// Mitsubishi GX Works2 project: A02_20251220_0   PLC: Q03UDV

TYPE Auto_Data : STRUCT
  Auto_Step : INT;  (* 自动流程字 *)
  Error_Code : INT;  (* 错误码 *)
  Task_Type : WORD;  (* 任务类型 *)
  Start_Row : INT;  (* 起点排 *)
  Start_Column : INT;  (* 起点列 *)
  Start_Layer : INT;  (* 起点层 *)
  End_Row : INT;  (* 终点排 *)
  End_Column : INT;  (* 终点列 *)
  End_Layer : INT;  (* 终点层 *)
  Picking_Station_No : INT;  (* 入库台编号 *)
  Placing_Station_No : INT;  (* 出库台编号 *)
  Task_Status : WORD;  (* 任务状态 *)
  Current_Task_ID : DWORD;  (* 当前任务ID *)
  Total_Number_Tasks : DINT;  (* 任务执行总次数 *)
  Stacker_Status : WORD;  (* 堆垛机状态 *)
  X_Current_Actual_Position : REAL;  (* X轴行走当前实际位置 *)
  Y_Current_Actual_Position : REAL;  (* Y轴升降当前实际位置 *)
  Z_Current_Actual_Position : REAL;  (* Z轴货叉当前实际位置 *)
  X_Current_Actual_Speed : REAL;  (* X轴行走当前实际速度 *)
  Y_Current_Actual_Speed : REAL;  (* Y轴升降当前实际速度 *)
  Z_Current_Actual_Speed : REAL;  (* Z轴货叉当前实际速度 *)
END_STRUCT END_TYPE

TYPE Axle_Data : STRUCT
  Auto_Target_Position : REAL;  (* Auto_目标位置 *)
  Auto_Positioning_Speed : REAL;  (* Auto_定位速度 *)
  Auto_Enable_Location : ARRAY [0..15] OF BOOL;  (* Auto_开启定位 *)
  Auto_Position_Reached : BOOL;  (* Auto_位置到达 *)
  Jog_Forward : BOOL;  (* 点动正转 *)
  Jog_Reverse : BOOL;  (* 点动反转 *)
  Forward_Enable : BOOL;  (* 正转允许 *)
  Reverse_Enable : BOOL;  (* 反转允许 *)
  o_wdCurrentPosition_F : REAL;  (* 当前位置 *)
  o_wdCurrentSpeed_F : REAL;  (* 当前速度 *)
  i_wdTargetPosition_F : REAL;  (* 目标位置 *)
  i_wdTargetVelocity_F : REAL;  (* 定位速度 *)
END_STRUCT END_TYPE

TYPE Pos : STRUCT
  X_Position : REAL;
  Y_Position : REAL;
  Z_Position : REAL;
END_STRUCT END_TYPE

TYPE Axle_attribute : STRUCT
  Motor_Actual_Position : REAL;  (* 电机实际位置 *)
  Position_Difference : REAL;  (* 位置差 *)
  Position_Reached : BOOL;  (* 位置到达 *)
END_STRUCT END_TYPE

TYPE Fork_Alarm : STRUCT
  Fork_Left_collapse_Alarm1 : BOOL;  (* 货叉左侧坍塌报警1 *)
  Fork_Left_collapse_Alarm2 : BOOL;  (* 货叉左侧坍塌报警2 *)
  Fork_Left_Width_Alarm1 : BOOL;  (* 货叉左超宽报警1 *)
  Fork_Left_Width_Alarm2 : BOOL;  (* 货叉左超宽报警2 *)
  Fork_Left_Height_Alarm : BOOL;  (* 货叉左侧超高报警 *)
  Fork_Right_collapse_Alarm1 : BOOL;  (* 货叉右侧坍塌报警1 *)
  Fork_Right_collapse_Alarm2 : BOOL;  (* 货叉右侧坍塌报警2 *)
  Fork_Right_Width_Alarm1 : BOOL;  (* 货叉右超宽报警1 *)
  Fork_Right_Width_Alarm2 : BOOL;  (* 货叉右超宽报警2 *)
  Fork_Right_Height_Alarm : BOOL;  (* 货叉右侧超高报警 *)
END_STRUCT END_TYPE

TYPE Sew_Write : STRUCT
  Control_Character : INT;  (* 控制字 *)
  Rated_Speed : INT;  (* 额定速度 *)
  Acceleration : INT;  (* 加速度 *)
  Deceleration : INT;  (* 减速度 *)
  Virtual_Input_Port : INT;  (* 虚拟输入端 *)
  Set_Mode : INT;  (* 设定应用模式 *)
  Target_Position : DINT;  (* 目标位置 *)
END_STRUCT END_TYPE

TYPE Sew_Read : STRUCT
  Status_Character : INT;  (* 状态字 *)
  Actual_Speed : INT;  (* 实际速度 *)
  Main_Status_Fault : WORD;  (* 状态主故障 *)
  Actual_Torque : INT;  (* 实际扭矩 *)
  Digital_Input_Port : INT;  (* 数字输入端 *)
  Actual_Mode : INT;  (* 实际应用模式 *)
  Actual_Position : DINT;  (* 实际位置 *)
END_STRUCT END_TYPE

TYPE Wcs_Data : STRUCT
  Task_Type : WORD;  (* 任务类型 *)
  Task_ID : DWORD;  (* 任务ID *)
  Start_Row : INT;  (* 起点排 *)
  Start_Column : INT;  (* 起点列 *)
  Start_Layer : INT;  (* 起点层 *)
  End_Row : INT;  (* 终点排 *)
  End_Column : INT;  (* 终点列 *)
  End_Layer : INT;  (* 终点层 *)
  Picking_Station_No : INT;  (* 入库台编号 *)
  Placing_Station_No : INT;  (* 出库台编号 *)
END_STRUCT END_TYPE

TYPE station_Status : STRUCT
  LoadGoods_Enable : BOOL;  (* 允许入库 *)
  UnLoadGoods_Enable : BOOL;  (* 允许出库 *)
END_STRUCT END_TYPE

TYPE manual_data : STRUCT
  X_ManualStart_Position : BOOL;  (* X轴单独定位 *)
  Y_ManualStart_Position : BOOL;  (* Y轴单独定位 *)
  Z_ManualStart_Position : BOOL;  (* Z轴单独定位 *)
  Position_Coords_Switch : BOOL;  (* 位置库位坐标切换 *)
  X_ManualPosition : REAL;  (* X轴定位位置 *)
  Y_ManualPosition : REAL;  (* Y轴定位位置 *)
  Z_ManualPosition : REAL;  (* Z轴定位位置 *)
  X_Manual_Column : INT;  (* X库位列 *)
  Y_Manual_Layer : INT;  (* Y库位层 *)
  X_ManualPosition_Assist : REAL;  (* X轴定位位置辅助 *)
  Y_ManualPosition_Assist : REAL;  (* Y轴定位位置辅助 *)
  Z_ManualPosition_Assist : REAL;  (* Z轴定位位置辅助 *)
  X_Manual_Column_Assist : INT;  (* X库位列辅助 *)
  Y_Manual_Layer_Assist : INT;  (* Y库位层辅助 *)
END_STRUCT END_TYPE

TYPE DInput : STRUCT
  AO2Safety_Circuit1 : BOOL;  (* AO2安全回路1 *)
  AO2Safety_Circuit2 : BOOL;  (* AO2安全回路2 *)
  Maintain_Run : BOOL;  (* 检修运行 *)
  Alarm_Reset : BOOL;  (* 故障复位 *)
  Admin : BOOL;  (* 管理者 *)
  Spare : BOOL;  (* 备用 *)
  Forward_Laser_Stop : BOOL;  (* 行走前方避障信号 *)
  Forward_Laser_Alarm : BOOL;  (* 行走前方避障故障 *)
  Reverse_Laser_Stop : BOOL;  (* 行走后方避障信号 *)
  Reverse_Laser_Alarm : BOOL;  (* 行走后方避障故障 *)
  Spare1 : BOOL;  (* 备用1 *)
  Spare2 : BOOL;  (* 备用2 *)
  Walk_Forward_TO_Pos : BOOL;  (* 行走前方限位 *)
  Walk_Reverse_TO_Pos : BOOL;  (* 行走后方限位 *)
  Walk_Deceleration : BOOL;  (* 行走减速 *)
  Spare3 : BOOL;  (* 备用3 *)
  Lift_Up_TO_Pos : BOOL;  (* 升降上限位 *)
  Lift_Down_TO_Pos : BOOL;  (* 升降下限位 *)
  Lift_Deceleration : BOOL;  (* 升降减速 *)
  Lift_Stall : BOOL;  (* 升降失速 *)
  Lift_Rope_Loosening1 : BOOL;  (* 升降松绳1 *)
  Lift_Rope_Loosening2 : BOOL;  (* 升降松绳2 *)
  Lift_Overload1 : BOOL;  (* 升降超重1 *)
  Lift_Overload2 : BOOL;  (* 升降超重2 *)
  Fork_Left_To_Pos : BOOL;  (* 伸缩左侧限位 *)
  Fork_Right_To_Pos : BOOL;  (* 伸缩右侧限位 *)
  Fork_Median_Detection1 : BOOL;  (* 伸缩中位检测1 *)
  Fork_Median_Detection2 : BOOL;  (* 伸缩中位检测2 *)
  Median_Goods_Detection : BOOL;  (* 中心物料检测 *)
  Walk_Drive_Power : BOOL;  (* 行走驱动器电源 *)
  Lift_Drive_Power : BOOL;  (* 升降驱动器电源 *)
  Fork_Drive_Power : BOOL;  (* 伸缩驱动器电源 *)
  Left_collapse_Signal1 : BOOL;  (* 左侧坍塌信号1 *)
  Left_collapse_Signal2 : BOOL;  (* 左侧坍塌信号2 *)
  Left_Width_Signal1 : BOOL;  (* 左侧超宽信号1 *)
  Left_Width_Signal2 : BOOL;  (* 左侧超宽信号2 *)
  Left_Height_Signal : BOOL;  (* 左侧超高检测 *)
  Left_Goods_Detection : BOOL;  (* 左侧物料检测 *)
  Spare4 : BOOL;  (* 备用4 *)
  Spare5 : BOOL;  (* 备用5 *)
  Right_collapse_Signal1 : BOOL;  (* 右侧坍塌信号1 *)
  Right_collapse_Signal2 : BOOL;  (* 右侧坍塌信号2 *)
  Right_Width_Signal1 : BOOL;  (* 右侧超宽信号1 *)
  Right_Width_Signal2 : BOOL;  (* 右侧超宽信号2 *)
  Right_Height_Signal : BOOL;  (* 右侧超高检测 *)
  Right_Goods_Detection : BOOL;  (* 右侧物料检测 *)
  Spare6 : BOOL;  (* 备用6 *)
  Spare7 : BOOL;  (* 备用7 *)
  Air_Error : BOOL;  (* 柜机空调故障 *)
  Optical_Error : BOOL;  (* 光通讯传感器故障 *)
  Spare8 : BOOL;  (* 备用8 *)
  Spare9 : BOOL;  (* 备用9 *)
  Walk_INV_Power : BOOL;  (* 行走变频器电源 *)
  Lift_INV_Power : BOOL;  (* 升降变频器电源 *)
  Fork_INV_Power : BOOL;  (* 伸缩变频器电源 *)
  Spare10 : BOOL;  (* 备用10 *)
  Console_Safety_Latch : BOOL;  (* 操作台安全插销 *)
  Spare11 : BOOL;  (* 备用11 *)
  Platform_Safety_Latch1 : BOOL;  (* 载货台安全插销1 *)
  Platform_Safety_Latch2 : BOOL;  (* 载货台安全插销2 *)
  Spare12 : BOOL;  (* 备用12 *)
  Spare13 : BOOL;  (* 备用13 *)
  Spare14 : BOOL;  (* 备用14 *)
  Spare15 : BOOL;  (* 备用15 *)
END_STRUCT END_TYPE

TYPE DOutput : STRUCT
  Pole_Light_R : BOOL;  (* 三色灯R *)
  Pole_Light_Y : BOOL;  (* 三色灯Y *)
  Pole_Light_G : BOOL;  (* 三色灯G *)
  Buzzer : BOOL;  (* 蜂鸣器 *)
  Walk_INV_Stop : BOOL;  (* 行走变频器停止 *)
  Lift_INV_Stop : BOOL;  (* 升降变频器停止 *)
  Fork_INV_Stop : BOOL;  (* 伸缩变频器停止 *)
  Spare5 : BOOL;  (* 备用5 *)
  Spare1 : BOOL;  (* 备用1 *)
  Spare2 : BOOL;  (* 备用2 *)
  Walk_Forward_Laser_Mode1 : BOOL;  (* 行走前方避障模式1 *)
  Walk_Forward_Laser_Mode2 : BOOL;  (* 行走前方避障模式2 *)
  Walk_Reverse_Laser_Mode1 : BOOL;  (* 行走后方避障模式1 *)
  Walk_Reverse_Laser_Mode2 : BOOL;  (* 行走后方避障模式2 *)
  Spare3 : BOOL;  (* 备用3 *)
  Spare4 : BOOL;  (* 备用4 *)
END_STRUCT END_TYPE

TYPE Sew_Status_Bit : STRUCT
  Ready_To_Run : BOOL;  (* 运行就绪 *)
  STO非活跃 : BOOL;  (* STO非活跃 *)
  输出级已使能 : BOOL;  (* 输出级已使能 *)
  制动器已打开 : BOOL;  (* 制动器已打开 *)
  电机旋转 : BOOL;  (* 电机旋转 *)
  Homed : BOOL;  (* 激活的驱动装置已寻参 *)
  已应用新的相对位置 : BOOL;  (* 已应用新的相对位置 *)
  Position_Arrive : BOOL;  (* 信息已就位激活 *)
  Error : BOOL;  (* 故障 *)
  警告 : BOOL;  (* 警告 *)
  驱动机构2激活 : BOOL;  (* 驱动机构2激活 *)
  消息额定_实际速度比较激活 : BOOL;  (* 消息额定_实际速度比较激活 *)
  软件限位开关非活跃 : BOOL;  (* 软件限位开关非活跃 *)
  预留 : BOOL;  (* 预留 *)
  待机运行激活 : BOOL;  (* 待机运行激活 *)
  HandshakeOut : BOOL;  (* HandshakeOut *)
END_STRUCT END_TYPE

TYPE Sew_Control_Bit : STRUCT
  Enable_Emergency_Stop : BOOL;  (* 使能紧急停止 *)
  Enable_Application_Stop : BOOL;  (* 使能应用停止 *)
  预留1 : BOOL;  (* 预留1 *)
  Brake_Open : BOOL;  (* 制动器释放 *)
  Forward_Jog : BOOL;  (* 正点动 *)
  Reverse_Jog : BOOL;  (* 负点动 *)
  接收相对位置 : BOOL;  (* 接收相对位置 *)
  Ramp_Bus_StartStop : BOOL;  (* 随总线斜波启动停止 *)
  Alarm_Reset : BOOL;  (* 故障复位 *)
  预留2 : BOOL;  (* 预留2 *)
  激活驱动机构2 : BOOL;  (* 激活驱动机构2 *)
  预留3 : BOOL;  (* 预留3 *)
  禁用软件限位开关 : BOOL;  (* 禁用软件限位开关 *)
  激活输出级锁定 : BOOL;  (* 激活输出级锁定 *)
  激活待机运行 : BOOL;  (* 激活待机运行 *)
  HandshakeIn : BOOL;  (* HandshakeIn *)
END_STRUCT END_TYPE

TYPE HMI : STRUCT
  Single_Mode_Switch : BOOL;  (* 自动单机模式 *)
  Manual_Mode_Switch : BOOL;  (* 手动模式 *)
  Maintenance_Mode_Switch : BOOL;  (* 维修模式 *)
  OnLine_Mode_Switch : BOOL;  (* 自动联机模式 *)
  Alarm_Reset : BOOL;  (* 报警复位 *)
  Single_RK_Type : BOOL;  (* 单机入库类型 *)
  Single_CK_Type : BOOL;  (* 单机出库类型 *)
  Single_YK_Type : BOOL;  (* 单机移库类型 *)
  OnLine_RK_Type : BOOL;  (* 联机入库类型 *)
  OnLine_CK_Type : BOOL;  (* 联机出库类型 *)
  OnLine_YK_Type : BOOL;  (* 联机移库类型 *)
  Auto_RK_Type : BOOL;  (* Auto入库类型 *)
  Auto_CK_Type : BOOL;  (* Auto出库类型 *)
  Auto_YK_Type : BOOL;  (* Auto移库类型 *)
  Continue_Task : BOOL;  (* 继续任务 *)
  End_Task : BOOL;  (* 终止任务 *)
  Pause_Task : BOOL;  (* 暂停任务 *)
  Laser_Close : BOOL;  (* 避障雷达关闭 *)
  Overload_Detection_Close : BOOL;  (* 超重检测关闭 *)
END_STRUCT END_TYPE

TYPE Master_R : STRUCT
  Stacker_Status : WORD;  (* 堆垛机状态 *)
  Auto_Step : INT;  (* 自动流程字 *)
  Error_Code : INT;  (* 错误码 *)
  Task_Status : WORD;  (* 任务状态 *)
  Current_Task_ID : DWORD;  (* 当前任务ID *)
  Total_Number_Tasks : DINT;  (* 任务执行总次数 *)
  X_Current_Actual_Position : INT;  (* 行走当前位置 *)
  Y_Current_Actual_Position : INT;  (* 升降当前位置 *)
  Z_Current_Actual_Position : INT;  (* 货叉当前位置 *)
  X_Current_Actual_Speed : INT;  (* 行走当前速度 *)
  Y_Current_Actual_Speed : INT;  (* 升降当前速度 *)
  Z_Current_Actual_Speed : INT;  (* 货叉当前速度 *)
  Current_Mode : INT;  (* 当前模式 *)
  Heartbeat : INT;  (* 心跳检测 *)
  LoadGoods_Apply : INT;  (* 取货请求 *)
  Spare : INT;  (* 无 *)
  UnLoadGoods_Apply : INT;  (* 卸货请求 *)
  Step_Record : INT;  (* 流程记录 *)
  X_Torque : INT;  (* X轴扭矩 *)
  Y_Torque : INT;  (* Y轴扭矩 *)
  Z_Torque : INT;  (* Z轴扭矩 *)
  X_Alarm_Code : WORD;  (* X轴报警 *)
  Y_Alarm_Code : WORD;  (* Y轴报警 *)
  Z_Alarm_Code : WORD;  (* Z轴报警 *)
  Stacker_Current_Column : INT;  (* 当前所在列 *)
  Stacker_Current_Layer : INT;  (* 当前所在层 *)
  Status_Bit : INT;  (* Status_Bit *)
  Warning_Code : INT;  (* 警告码 *)
END_STRUCT END_TYPE

TYPE Master_W : STRUCT
  Task_Type : WORD;  (* 任务类型 *)
  Task_ID : DWORD;  (* 任务ID *)
  Start_Column : INT;  (* 起点列 *)
  Start_Row : INT;  (* 起点排 *)
  Start_Layer : INT;  (* 起点层 *)
  End_Column : INT;  (* 终点列 *)
  End_Row : INT;  (* 终点排 *)
  End_Layer : INT;  (* 终点层 *)
  Placing_Station_No : INT;  (* 出库台编号 *)
  Picking_Station_No : INT;  (* 入库台编号 *)
  Heartbeat : INT;  (* 系统心跳 *)
  LoadGoods_Enable_B1 : INT;  (* 允许取货B01 *)
  LoadGoods_Enable_B2 : INT;  (* 允许取货B02 *)
  UnLoadGoods_Enable_B2 : INT;  (* 允许放货B02 *)
  UnLoadGoods_Enable_B1 : INT;  (* 允许放货B01 *)
  Reset_Control : INT;  (* 复位控制 *)
  Mode_Switch : INT;  (* Mode *)
  Pause_Control : INT;  (* 暂停控制 *)
  Y_Locate_Position : INT;  (* Y轴定位位置 *)
  X_Locate_Position : INT;  (* X轴定位位置 *)
  Z_Locate_Position : INT;  (* Z轴定位位置 *)
  X_Locate_Column : INT;  (* X轴定位列 *)
  Y_Locate_Layer : INT;  (* Y轴定位层 *)
  EStop_Control : INT;  (* 紧急停止 *)
  Spare16 : INT;  (* 备用16 *)
  Spare17 : INT;  (* 备用17 *)
  Spare18 : INT;  (* 备用18 *)
  Spare19 : INT;  (* 备用19 *)
  Control_Bit : INT;  (* Control_Bit *)
END_STRUCT END_TYPE

TYPE parameter : STRUCT
  X_Auto_Speed : INT;  (* X轴自动速度设置 *)
  Y_Auto_Speed : INT;  (* Y轴自动速度设置 *)
  Z_Auto_Speed : INT;  (* Z轴自动速度设置 *)
  X_Manual_Speed : INT;  (* X轴手动速度设置 *)
  Y_Manual_Speed : INT;  (* Y轴手动速度设置 *)
  Z_Manual_Speed : INT;  (* Z轴手动速度设置 *)
  X_LimitPos : REAL;  (* X轴前限位设置 *)
  X_NegativePos : REAL;  (* X轴后限位设置 *)
  Y_LimitPos : REAL;  (* Y轴上限位设置 *)
  Y_NegativePos : REAL;  (* Y轴下限位设置 *)
  Z_LimitPos : REAL;  (* Z轴左限位设置 *)
  Z_NegativePos : REAL;  (* Z轴右限位设置 *)
  X_OffsetPos : REAL;  (* X轴位置偏移设置 *)
  Y_OffsetPos : REAL;  (* Y轴位置偏移设置 *)
  Z_OffsetPos : REAL;  (* Z轴位置偏移设置 *)
  X_Acceleration : INT;  (* X轴加速度 *)
  X_Deceleration : INT;  (* X轴减速度 *)
  Y_Acceleration : INT;  (* Y轴加速度 *)
  Y_Deceleration : INT;  (* Y轴减速度 *)
  Z_Acceleration : INT;  (* Z轴加速度 *)
  Z_Deceleration : INT;  (* Z轴减速度 *)
  Y_LoadGoods_Speed : INT;  (* Y轴取放物料速度 *)
END_STRUCT END_TYPE

TYPE laser : STRUCT
  前方避障停止检测 : BOOL;  (* 前方避障停止检测 *)
  后方避障减速检测 : BOOL;  (* 后方避障减速检测 *)
  前方避障减速检测 : BOOL;  (* 前方避障减速检测 *)
  后方避障停止检测 : BOOL;  (* 后方避障停止检测 *)
  Obstacle_Alarm : BOOL;  (* 激光避障报警 *)
END_STRUCT END_TYPE

TYPE record : STRUCT
  Task_Type : WORD;  (* 任务类型 *)
  Start_Row : INT;  (* 起点排 *)
  Start_Column : INT;  (* 起点列 *)
  Start_Layer : INT;  (* 起点层 *)
  End_Row : INT;  (* 终点排 *)
  End_Column : INT;  (* 终点列 *)
  End_Layer : INT;  (* 终点层 *)
  Picking_Station_No : INT;  (* 入库台编号 *)
  Placing_Station_No : INT;  (* 出库台编号 *)
  Auto_Step : INT;  (* 自动流程字 *)
  Current_Task_ID : DWORD;  (* 当前任务ID *)
END_STRUCT END_TYPE

TYPE Stacker_R_Status_Bit : STRUCT
  Stacker_A01ManualControl : BOOL;  (* 堆垛机地面手动控制中 *)
  Advance_To_Position : BOOL;  (* 前进到位 *)
  Retreat_To_Position : BOOL;  (* 后退到位 *)
  Ascend_To_Position : BOOL;  (* 上升到位 *)
  Descend_To_Position : BOOL;  (* 下降到位 *)
  Left_To_Position : BOOL;  (* 左伸到位 *)
  Right_To_Position : BOOL;  (* 右伸到位 *)
  Fork_Zero : BOOL;  (* 货叉在中位 *)
  Picked_Up : BOOL;  (* 取货中 *)
  Releasing_Goods : BOOL;  (* 放货中 *)
  Spare3 : BOOL;  (* 备用3 *)
  Spare4 : BOOL;  (* 备用4 *)
  Spare5 : BOOL;  (* 备用5 *)
  Spare6 : BOOL;  (* 备用6 *)
  Spare7 : BOOL;  (* 备用7 *)
  Spare8 : BOOL;  (* 备用8 *)
END_STRUCT END_TYPE

TYPE Stacker_W_Control_Bit : STRUCT
  Apply_Manual_Control : BOOL;  (* 请求手动控制 *)
  Position_Coords_Switch : BOOL;  (* 位置库位定位切换 *)
  X_ManualStart_Position : BOOL;  (* X轴定位 *)
  Y_ManualStart_Position : BOOL;  (* Y轴定位 *)
  Z_ManualStart_Position : BOOL;  (* Z轴定位 *)
  X_Jog_Forward : BOOL;  (* X轴前进 *)
  X_Jog_Reverse : BOOL;  (* X轴后退 *)
  Y_Jog_Forward : BOOL;  (* Y轴上升 *)
  Y_Jog_Reverse : BOOL;  (* Y轴下降 *)
  Z_Jog_Forward : BOOL;  (* Z轴左伸 *)
  Z_Jog_Reverse : BOOL;  (* Z轴右伸 *)
  Manual_Y_Force_Enable : BOOL;  (* Y轴强制动作 *)
  End_Task : BOOL;  (* 终止任务 *)
  Continue_Task : BOOL;  (* 继续任务 *)
  Spare3 : BOOL;  (* 备用3 *)
  Spare4 : BOOL;  (* 备用4 *)
  Spare5 : BOOL;  (* 备用5 *)
  Spare6 : BOOL;  (* 备用6 *)
END_STRUCT END_TYPE

// global labels: Global1
VAR_GLOBAL
  Auto_Data : Auto_Data;
  Auto_Run AT M500 : BOOL;  (* 自动运行中 *)
  Auto_Run_Conditions AT M501 : BOOL;  (* 自动运行条件 *)
  OnLine_Mode AT M502 : BOOL;  (* 自动联机模式状态 *)
  Manual_Mode AT M504 : BOOL;  (* 手动模式状态 *)
  Maintenance_Mode AT M505 : BOOL;  (* 维修模式状态 *)
  Fork_Zero AT M506 : BOOL;  (* Fork_在零点 *)
  Fork_Load_Done AT M507 : BOOL;  (* Fork_取料完成 *)
  Fork_Unload_Done AT M508 : BOOL;  (* Fork_放料完成 *)
  Resetting_Alarm : BOOL;  (* 报警复位中 *)
  Coords_Home : BOOL;  (* 库位校零 *)
  Height_Goods_Lifted : REAL;  (* 货物抬起高度设置 *)
  Wcs_interface : Wcs_Data;
  Fork_Goods_Detection : ARRAY [0..1] OF BOOL;  (* Fork探货检测 *)
  Manual : manual_data;
  Axle_attribute : ARRAY [0..2] OF Axle_attribute;  (* 轴属性 *)
  Stacker_Current_Column AT D400 : INT;  (* 堆垛机当前所在列 *)
  Stacker_Current_Layer AT D402 : INT;  (* 堆垛机当前所在层 *)
  Mode AT D404 : INT;  (* 0联机 1单机 2手动 3维修 *)
  Platform_Goods_Detection : BOOL;  (* 货叉物料检测 *)
  Stacker_Stationary : BOOL;  (* 堆垛机静止中 *)
  Alone : Wcs_Data;
  E_Stop : BOOL;  (* 急停开关 *)
  Single_Mode AT M503 : BOOL;  (* 自动单机模式状态 *)
  Fork_Alarm : Fork_Alarm;
  Laser : laser;
  Language_Switch AT M700 : BOOL;  (* 语言切换 *)
  Language AT D5030 : INT;  (* 语言显示 *)
  Password AT D5032 : INT;  (* 密码权限 *)
  Mode_Record : INT;  (* 模式记录 *)
  Alarm_record AT M800 : ARRAY [1..48] OF BOOL;
  Positioning_Enable : ARRAY [0..2] OF BOOL;  (* 定位允许 *)
  Record : record;  (* 任务记录 *)
  Fork_Middle_Detection AT M701 : BOOL;  (* 货叉伸缩中位检测 *)
  Manual_Y_Force_Enable AT M702 : BOOL;  (* 手动Y轴强制允许 *)
  Height_Goods_Lowered : REAL;  (* 货物下降高度设置 *)
  Warning_Code AT D406 : INT;
  HMI_Screen AT D407 : INT;  (* HMI画面 *)
  Screen_Assistance : BOOL;  (* 弹窗辅助 *)
  Maintenance_Mode_Stop : BOOL;  (* 维修模式断开 *)
END_VAR

// global labels: Coords
VAR_GLOBAL
  Column_Coords : ARRAY [1..14] OF REAL;  (* 列坐标 *)
  Layer_Coords : ARRAY [1..5] OF REAL;  (* 层坐标 *)
  Row_Coords : ARRAY [1..2] OF REAL;  (* 排坐标 *)
  Station_Coords : ARRAY [0..4] OF Pos;  (* 对接台坐标 *)
  Station_Status : ARRAY [0..4] OF station_Status;  (* 对接台状态 *)
END_VAR

// global labels: Drive
VAR_GLOBAL
  Axle_X_Sew_Read : Sew_Read;
  Axle_X_Sew_Write : Sew_Write;
  Axle_Y_Sew_Read : Sew_Read;
  Axle_Z_Sew_Read : Sew_Read;
  Axle_Y_Sew_Write : Sew_Write;
  Axle_Z_Sew_Write : Sew_Write;
  Axle : ARRAY [0..2] OF Axle_Data;
  Axle_X_Sew_Status_Bit : Sew_Status_Bit;
  Axle_Y_Sew_Status_Bit : Sew_Status_Bit;
  Axle_Z_Sew_Status_Bit : Sew_Status_Bit;
  Axle_X_Sew_Control_Bit : Sew_Control_Bit;
  Axle_Y_Sew_Control_Bit : Sew_Control_Bit;
  Axle_Z_Sew_Control_Bit : Sew_Control_Bit;
  Axle_X_Status AT D180 : WORD;
  Axle_Y_Status AT D181 : WORD;
  Axle_Z_Status AT D182 : WORD;
  Axle_X_Alalm AT D183 : WORD;
  Axle_Y_Alalm AT D184 : WORD;
  Axle_Z_Alalm AT D185 : WORD;
END_VAR

// global labels: IO
VAR_GLOBAL
  DInput : DInput;
  DOutput : DOutput;
END_VAR

// global labels: HMI
VAR_GLOBAL
  HMI : HMI;
  Parameter_Set : parameter;
END_VAR

// global labels: Master
VAR_GLOBAL
  Master_R : Master_R;
  Master_W : Master_W;
  Stacker_W_Control_Bit : Stacker_W_Control_Bit;
  Stacker_R_Status_Bit : Stacker_R_Status_Bit;
END_VAR

PROGRAM MAIN
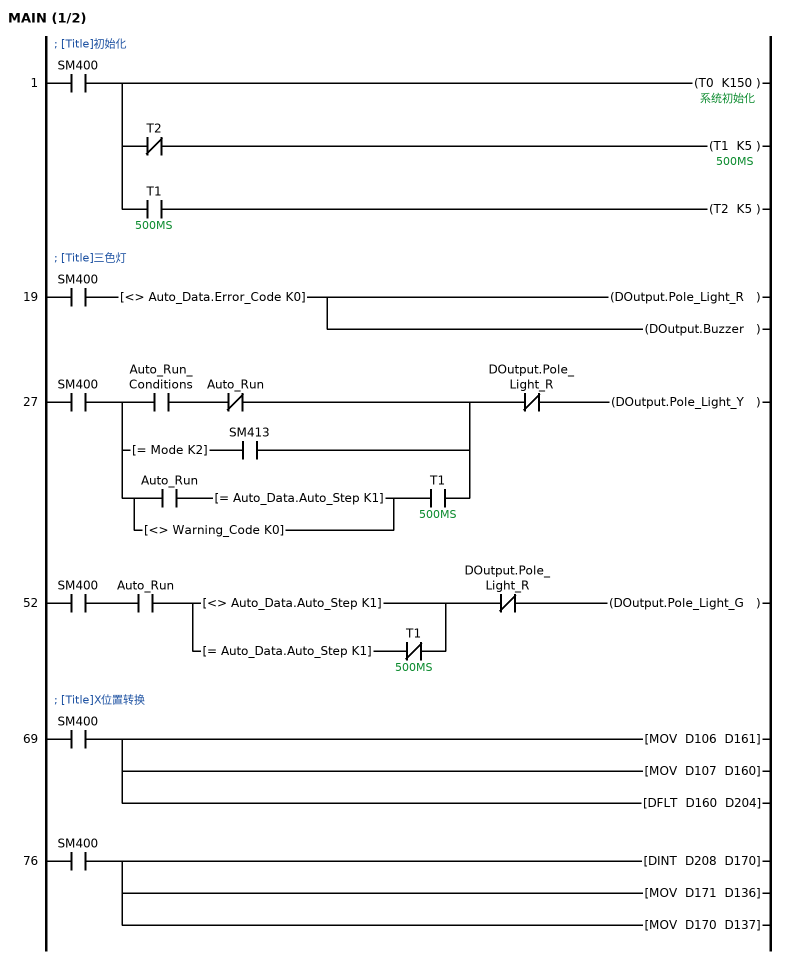
; [Title]初始化
1     LD      SM400
      OUT     T0 K150  ; 系统初始化
      MPS
      ANI     T2
      OUT     T1 K5  ; 500MS
      MPP
      AND     T1  ; 500MS
      OUT     T2 K5
; [Title]三色灯
19    LD      SM400
      AND<>   Auto_Data.Error_Code K0
      OUT     DOutput.Pole_Light_R
      OUT     DOutput.Buzzer
27    LD      SM400
      LD      Auto_Run_Conditions
      ANI     Auto_Run
      LD=     Mode K2
      AND     SM413
      ORB
      LD      Auto_Run
      AND=    Auto_Data.Auto_Step K1
      OR<>    Warning_Code K0
      AND     T1  ; 500MS
      ORB
      ANB
      ANI     DOutput.Pole_Light_R
      OUT     DOutput.Pole_Light_Y
52    LD      SM400
      AND     Auto_Run
      LD<>    Auto_Data.Auto_Step K1
      LD=     Auto_Data.Auto_Step K1
      ANI     T1  ; 500MS
      ORB
      ANB
      ANI     DOutput.Pole_Light_R
      OUT     DOutput.Pole_Light_G
; [Title]X位置转换
69    LD      SM400
      MOV     D106 D161
      MOV     D107 D160
      DFLT    D160 D204
76    LD      SM400
      DINT    D208 D170
      MOV     D171 D136
      MOV     D170 D137
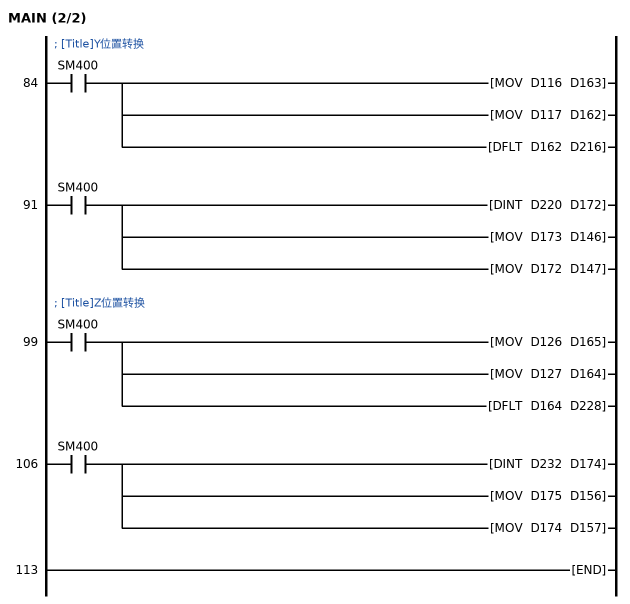
; [Title]Y位置转换
84    LD      SM400
      MOV     D116 D163
      MOV     D117 D162
      DFLT    D162 D216
91    LD      SM400
      DINT    D220 D172
      MOV     D173 D146
      MOV     D172 D147
; [Title]Z位置转换
99    LD      SM400
      MOV     D126 D165
      MOV     D127 D164
      DFLT    D164 D228
106   LD      SM400
      DINT    D232 D174
      MOV     D175 D156
      MOV     D174 D157
113   END
END_PROGRAM

PROGRAM 05_Study
VAR
  AO : INT;
END_VAR
(*列间距:=1870;
层间距:=875;
总列数:=14;
总层数:=5;*)

Row_Coords[1]:=-1970.0;
Row_Coords[2]:=1970.0;

IF Column_Coords[1] =0.0 AND Layer_Coords[1] =0.0  THEN
	FOR AO:=1 TO 13 DO
	Column_Coords[AO+1]:=Column_Coords[AO] +1870.0;
    END_FOR;
END_IF;

Layer_Coords[1]:=0.0;
Layer_Coords[2]:=900.0;
Layer_Coords[3]:=1800.0;
Layer_Coords[4]:=2925.0;
Layer_Coords[5]:=3825.0;
END_PROGRAM

PROGRAM 06_Auto
(*参数设置MM*)
Height_Goods_Lifted:=60.0;
Height_Goods_Lowered:=40.0;

(*非自动模式*)
IF Mode>1 THEN
	Auto_Data.Auto_Step:=0;
	Auto_Run := FALSE;
END_IF;

(*初始化*)
IF Auto_Data.Auto_Step=0 THEN
	Fork_Load_Done:=FALSE;
	Fork_Unload_Done:=FALSE;
	Auto_Data.Picking_Station_No:=0;
	Auto_Data.Placing_Station_No:=0;
	Auto_Data.Task_Type:=0;
	Auto_Data.Start_Row:=0;
	Auto_Data.Start_Column:=0;
	Auto_Data.Start_Layer:=0;
	Auto_Data.End_Row:=0;
	Auto_Data.End_Column:=0;
	Auto_Data.End_Layer:=0;
	Auto_Run := FALSE;
	Master_R.LoadGoods_Apply:=0;
	Master_R.UnLoadGoods_Apply:=0;
	Stacker_R_Status_Bit.Picked_Up:=FALSE;
	Stacker_R_Status_Bit.Releasing_Goods:=FALSE;
	Axle[0].Auto_Enable_Location[1]:=FALSE;
	Axle[1].Auto_Enable_Location[1]:=FALSE;
	Axle[2].Auto_Enable_Location[1]:=FALSE;
END_IF;

(*自动运行条件*)
IF Auto_Data.Auto_Step=0 AND Auto_Run=FALSE AND Mode<=1 AND E_Stop=FALSE AND Resetting_Alarm=FALSE AND TS0  AND
    Axle_X_Sew_Status_Bit.Ready_To_Run AND Axle_Y_Sew_Status_Bit.Ready_To_Run AND Axle_Z_Sew_Status_Bit.Ready_To_Run AND 
    Axle_X_Sew_Status_Bit.Error=FALSE AND Axle_Y_Sew_Status_Bit.Error=FALSE AND Axle_Z_Sew_Status_Bit.Error=FALSE AND 
    Axle_X_Sew_Status_Bit.Homed AND Axle_Y_Sew_Status_Bit.Homed AND Axle_Z_Sew_Status_Bit.Homed AND 
	 Auto_Data.Error_Code=0 THEN
	Auto_Run_Conditions:=TRUE;
ELSE
	Auto_Run_Conditions:=FALSE;
END_IF;

(*堆垛机状态*)
Auto_Data.Stacker_Status:=0;
IF Auto_Data.Auto_Step=0 AND Auto_Run=FALSE AND Mode<=1 AND Auto_Run_Conditions THEN
	Auto_Data.Stacker_Status:=1;
END_IF;
IF  Auto_Data.Auto_Step<>0 OR Auto_Run  THEN
	Auto_Data.Stacker_Status:=2;
END_IF;
IF Auto_Data.Error_Code<>0 THEN
	Auto_Data.Stacker_Status:=3;
END_IF;

(*任务开始 WCS就绪---联机模式*) (*Mode_ 0联机 1单机 2手动 3维修*)
IF Auto_Data.Stacker_Status=1 AND  Wcs_interface.Task_ID <> 0 THEN
	(*入库*)
	    IF Wcs_interface.Task_Type = 1 AND Wcs_interface.Task_ID <> Auto_Data.Current_Task_ID  AND Wcs_interface.Picking_Station_No<>0 AND 
			(Wcs_interface.End_Row<>0 AND Wcs_interface.End_Column<>0 AND Wcs_interface.End_Layer<>0)  AND Mode=0 AND
            Auto_Data.Auto_Step = 0 AND Auto_Run = FALSE THEN
    
                  Auto_Run := TRUE;
                  Auto_Data.Current_Task_ID:= Wcs_interface.Task_ID;
				  Auto_Data.Task_Type:= Wcs_interface.Task_Type;
				  Auto_Data.Picking_Station_No:= Wcs_interface.Picking_Station_No;
				  Auto_Data.End_Row:= Wcs_interface.End_Row;
				  Auto_Data.End_Column:= Wcs_interface.End_Column;
				  Auto_Data.End_Layer:= Wcs_interface.End_Layer;
				  Auto_Data.Total_Number_Tasks := Auto_Data.Total_Number_Tasks+1;
				  Auto_Data.Task_Status:=1;
				  Auto_Data.Auto_Step:=1;
		END_IF;
		
		(*出库*)
		IF Wcs_interface.Task_Type = 2 AND Wcs_interface.Task_ID <> Auto_Data.Current_Task_ID AND Wcs_interface.Placing_Station_No<>0 AND 
			(Wcs_interface.Start_Row<>0 AND Wcs_interface.Start_Column<>0 AND Wcs_interface.Start_Layer<>0) AND Mode=0 AND
            Auto_Data.Auto_Step = 0 AND Auto_Run = FALSE THEN
    
			Auto_Run := TRUE;
			Auto_Data.Current_Task_ID:= Wcs_interface.Task_ID;
			Auto_Data.Task_Type:= Wcs_interface.Task_Type;
			Auto_Data.Placing_Station_No:= Wcs_interface.Placing_Station_No;
			Auto_Data.Start_Row:= Wcs_interface.Start_Row;
			Auto_Data.Start_Column:= Wcs_interface.Start_Column;
			Auto_Data.Start_Layer:= Wcs_interface.Start_Layer;
			Auto_Data.Total_Number_Tasks := Auto_Data.Total_Number_Tasks+1;
			Auto_Data.Task_Status:=2;
			 Auto_Data.Auto_Step:=1;
		END_IF;
		
		(*移库*)
		IF Wcs_interface.Task_Type = 3 AND Wcs_interface.Task_ID <> Auto_Data.Current_Task_ID  AND Mode=0 AND
			(Wcs_interface.Start_Row<>0 AND Wcs_interface.Start_Column<>0 AND Wcs_interface.Start_Layer<>0 AND Wcs_interface.End_Row<>0 AND Wcs_interface.End_Column<>0 AND Wcs_interface.End_Layer<>0 )AND 
            Auto_Data.Auto_Step = 0 AND Auto_Run = FALSE THEN
    
			Auto_Run := TRUE;
			Auto_Data.Current_Task_ID:= Wcs_interface.Task_ID;
			Auto_Data.Task_Type:= Wcs_interface.Task_Type;
			Auto_Data.Start_Row:= Wcs_interface.Start_Row;
			Auto_Data.Start_Column:= Wcs_interface.Start_Column;
			Auto_Data.Start_Layer:= Wcs_interface.Start_Layer;
			Auto_Data.End_Row:= Wcs_interface.End_Row;
			Auto_Data.End_Column:= Wcs_interface.End_Column;
			Auto_Data.End_Layer:= Wcs_interface.End_Layer;
			Auto_Data.Total_Number_Tasks := Auto_Data.Total_Number_Tasks+1;
			Auto_Data.Task_Status:=3;
			 Auto_Data.Auto_Step:=1;
		END_IF;
		
		(*回检修位置*)
		IF Wcs_interface.Task_Type = 4 AND Wcs_interface.Task_ID <> Auto_Data.Current_Task_ID AND Mode=0 AND 
			 Wcs_interface.Start_Row=0 AND Wcs_interface.Start_Column=0 AND Wcs_interface.Start_Layer=0 AND Wcs_interface.End_Row=0 AND Wcs_interface.End_Column=0 AND Wcs_interface.End_Layer=0 AND 
            Wcs_interface.Picking_Station_No=0 AND Wcs_interface.Placing_Station_No=0 AND Auto_Data.Auto_Step = 0 AND Auto_Run = FALSE THEN
            Auto_Run := TRUE;
			Auto_Data.Current_Task_ID:= Wcs_interface.Task_ID;
			Auto_Data.Task_Type:= Wcs_interface.Task_Type;
			Auto_Data.Task_Status:=4;
            Auto_Data.Auto_Step:=1;
		END_IF;
END_IF;

(*非单机模式*)
IF Mode<>1 THEN
	Alone.Task_Type :=0;
	Alone.Task_ID :=0;
END_IF;

(*任务开始 WCS就绪---单机模式*) (*Mode_ 0联机 1单机 2手动 3维修*)
IF Auto_Data.Stacker_Status=1 AND Alone.Task_ID <>0 THEN
	(*入库*)
	    IF Alone.Task_Type = 1 AND Alone.Task_ID <> Auto_Data.Current_Task_ID AND Alone.Picking_Station_No<>0 AND 
			(Alone.End_Row<>0 AND Alone.End_Column<>0 AND Alone.End_Layer<>0)  AND Mode=1 AND
            Auto_Data.Auto_Step = 0 AND Auto_Run = FALSE THEN
    
                  Auto_Run := TRUE;
                  Auto_Data.Current_Task_ID:= Alone.Task_ID;
				  Auto_Data.Task_Type:= Alone.Task_Type;
				  Auto_Data.Picking_Station_No:= Alone.Picking_Station_No;
				  Auto_Data.End_Row:= Alone.End_Row;
				  Auto_Data.End_Column:= Alone.End_Column;
				  Auto_Data.End_Layer:= Alone.End_Layer;
				  Auto_Data.Total_Number_Tasks := Auto_Data.Total_Number_Tasks+1;
				  Auto_Data.Task_Status:=1;
				   Auto_Data.Auto_Step:=1;
		END_IF;
		
		(*出库*)
		IF Alone.Task_Type = 2 AND Alone.Task_ID <> Auto_Data.Current_Task_ID AND Alone.Placing_Station_No<>0 AND 
			(Alone.Start_Row<>0 AND Alone.Start_Column<>0 AND Alone.Start_Layer<>0) AND Mode=1 AND
            Auto_Data.Auto_Step = 0 AND Auto_Run = FALSE THEN
    
			Auto_Run := TRUE;
			Auto_Data.Current_Task_ID:= Alone.Task_ID;
			Auto_Data.Task_Type:= Alone.Task_Type;
			Auto_Data.Placing_Station_No:= Alone.Placing_Station_No;
			Auto_Data.Start_Row:= Alone.Start_Row;
			Auto_Data.Start_Column:= Alone.Start_Column;
			Auto_Data.Start_Layer:= Alone.Start_Layer;
			Auto_Data.Total_Number_Tasks := Auto_Data.Total_Number_Tasks+1;
			Auto_Data.Task_Status:=2;
			 Auto_Data.Auto_Step:=1;
		END_IF;
		
		(*移库*)
		IF Alone.Task_Type = 3 AND Alone.Task_ID <> Auto_Data.Current_Task_ID  AND Mode=1 AND
			(Alone.Start_Row<>0 AND Alone.Start_Column<>0 AND Alone.Start_Layer<>0 AND Alone.End_Row<>0 AND Alone.End_Column<>0 AND Alone.End_Layer<>0 )AND 
            Auto_Data.Auto_Step = 0 AND Auto_Run = FALSE THEN
    
			Auto_Run := TRUE;
			Auto_Data.Current_Task_ID:= Alone.Task_ID;
			Auto_Data.Task_Type:= Alone.Task_Type;
			Auto_Data.Start_Row:= Alone.Start_Row;
			Auto_Data.Start_Column:= Alone.Start_Column;
			Auto_Data.Start_Layer:= Alone.Start_Layer;
			Auto_Data.End_Row:= Alone.End_Row;
			Auto_Data.End_Column:= Alone.End_Column;
			Auto_Data.End_Layer:= Alone.End_Layer;
			Auto_Data.Total_Number_Tasks := Auto_Data.Total_Number_Tasks+1;
			Auto_Data.Task_Status:=3;
			 Auto_Data.Auto_Step:=1;
		END_IF;
		
		(*回检修位置*)
		IF Alone.Task_Type = 4 AND Alone.Task_ID <> Auto_Data.Current_Task_ID AND Mode=1 AND 
			 Alone.Start_Row=0 AND Alone.Start_Column=0 AND Alone.Start_Layer=0 AND Alone.End_Row=0 AND Alone.End_Column=0 AND Alone.End_Layer=0 AND 
            Alone.Picking_Station_No=0 AND Alone.Placing_Station_No=0 AND Auto_Data.Auto_Step = 0 AND Auto_Run = FALSE THEN
            Auto_Run := TRUE;
			Auto_Data.Current_Task_ID:= Alone.Task_ID;
			Auto_Data.Task_Type:= Alone.Task_Type;
			Auto_Data.Task_Status:=4;
            Auto_Data.Auto_Step:=1;
		END_IF;
END_IF;

(*任务纪录*)
IF Auto_Data.Auto_Step=1 THEN
    Record.Current_Task_ID:=Auto_Data.Current_Task_ID;
    Record.Task_Type:=Auto_Data.Task_Type;
    Record.Start_Row:=Auto_Data.Start_Row;
    Record.Start_Column:=Auto_Data.Start_Column;
    Record.Start_Layer:=Auto_Data.Start_Layer;
    Record.End_Row:=Auto_Data.End_Row;
    Record.End_Column:=Auto_Data.End_Column;
    Record.End_Layer:=Auto_Data.End_Layer;
    Record.Picking_Station_No:=Auto_Data.Picking_Station_No;
    Record.Placing_Station_No:=Auto_Data.Placing_Station_No;
END_IF;
(*流程纪录*)
IF Auto_Data.Auto_Step<>0 AND Record.Auto_Step<>Auto_Data.Auto_Step THEN
	Record.Auto_Step:=Auto_Data.Auto_Step;
END_IF;
 
(*延时2秒开始自动流程*)
OUT_T(Auto_Run AND Auto_Data.Auto_Step=1,TC17,20);
IF TS17 THEN
	Auto_Data.Auto_Step:=2;
	rst(TS17,TC17);
END_IF;

(*任务失败*)
IF Auto_Data.Auto_Step <> 0 AND Auto_Data.Error_Code <> 0  THEN
	Auto_Data.Task_Status:=6;
    Auto_Run := FALSE;
	Axle[0].Auto_Enable_Location[1]:=FALSE;
	Axle[1].Auto_Enable_Location[1]:=FALSE;
	Axle[2].Auto_Enable_Location[1]:=FALSE;
END_IF;

(*继续任务*)
IF (HMI.Continue_Task OR Stacker_W_Control_Bit.Continue_Task) AND Record.Auto_Step<>0 AND Auto_Data.Stacker_Status=1 AND  Auto_Data.Error_Code=0 THEN
	HMI.Pause_Task:=FALSE;
	Auto_Data.Current_Task_ID:= Record.Current_Task_ID;
	Auto_Data.Task_Type:= Record.Task_Type;
	Auto_Data.Picking_Station_No:= Record.Picking_Station_No;
	Auto_Data.Placing_Station_No:= Record.Placing_Station_No;
    Auto_Data.Start_Row:= Record.Start_Row;
	Auto_Data.Start_Column:= Record.Start_Column;
	Auto_Data.Start_Layer:= Record.Start_Layer;
	Auto_Data.End_Row:=  Record.End_Row;
	Auto_Data.End_Column:= Record.End_Column;
	Auto_Data.End_Layer:= Record.End_Layer;
	Auto_Data.Auto_Step:=Record.Auto_Step;
	Auto_Run := TRUE;
	Auto_Data.Total_Number_Tasks := Auto_Data.Total_Number_Tasks+1;
END_IF;

(*终止任务*)
IF (HMI .End_Task OR Stacker_W_Control_Bit.End_Task) AND (Auto_Data.Auto_Step<>0 OR Record.Auto_Step<>0)   THEN
	        HMI.Pause_Task:=FALSE;
			Alone.Picking_Station_No:=0;
			Alone.Placing_Station_No:=0;
			Alone.Task_Type:=0;
			Alone.Start_Row:=0;
			Alone.Start_Column:=0;
			Alone.Start_Layer:=0;
			Alone.End_Row:=0;
			Alone.End_Column:=0;
			Alone.End_Layer:=0;
			Auto_Data.Task_Status:=7;
			Auto_Data.Auto_Step:=0;
			Auto_Run := FALSE;
			Record.Auto_Step:=0	;	
END_IF;
	
(*自动流程开始*)
IF Auto_Run AND Auto_Data.Error_Code=0 AND HMI.Pause_Task=FALSE AND Master_W.Pause_Control<>1THEN
  CASE Auto_Data.Auto_Step OF
	2:  (*货叉是否在零位*)
	    IF Fork_Zero=FALSE THEN
	         Axle[2].Auto_Target_Position:=0.0;
		     Axle[2].Auto_Enable_Location[1]:=TRUE;
		END_IF;
		 
          IF Fork_Zero THEN
			   Axle[2].Auto_Enable_Location[1]:=FALSE;
                 IF Auto_Data.Task_Type>=1 AND Auto_Data.Task_Type<=4 THEN
			          Auto_Data.Auto_Step:=3;
			     END_IF;
		END_IF;

	3: (*入库 *)
		 IF Auto_Data.Task_Type=1   AND Auto_Data.Picking_Station_No<>0 AND 
			 Auto_Data.End_Row<>0 AND Auto_Data.End_Column<>0 AND Auto_Data.End_Layer<>0 THEN
			 IF Platform_Goods_Detection THEN 
			        Auto_Data.Auto_Step:=15;     (*入库任务 载货台有料 前往终点库位*)
			 ELSE
			   Auto_Data.Auto_Step:=10;
			 END_IF;
		 END_IF;
		 
		(*出库 移库*)
		IF ((Auto_Data.Task_Type=2   AND Auto_Data.Placing_Station_No<>0 ) OR (Auto_Data.Task_Type=3 AND Auto_Data.End_Row<>0 AND Auto_Data.End_Column<>0 AND Auto_Data.End_Layer<>0)) AND
			Auto_Data.Start_Row<>0 AND Auto_Data.Start_Column<>0 AND Auto_Data.Start_Layer<>0 THEN
			IF Platform_Goods_Detection THEN
				IF Auto_Data.Task_Type=3 OR Auto_Data.Task_Type=2 THEN
			        Auto_Data.Auto_Step:=15;     (*移库任务  载货台有料 前往终点库位*)
				END_IF;
			ELSE
			Auto_Data.Auto_Step:=10;
			END_IF;	
		END_IF;	
		
		(*回检修位置*)
		IF Auto_Data.Task_Type=4    THEN
			Auto_Data.Auto_Step:=10;
		END_IF;	
  END_CASE; 
END_IF;
		

IF Auto_Run AND Auto_Data.Error_Code=0  AND HMI.Pause_Task=FALSE AND Master_W.Pause_Control<>1 THEN
	CASE Auto_Data.Auto_Step OF
    10:  (*前往取货点*)
         IF Auto_Data.Task_Type=1  THEN
         	   Axle[0].Auto_Target_Position:=Station_Coords[ Auto_Data.Picking_Station_No].X_Position;
			   Axle[1].Auto_Target_Position:=Station_Coords[ Auto_Data.Picking_Station_No].Y_Position-Height_Goods_Lifted;
			   Axle[0].Auto_Enable_Location[1]:=TRUE;
			   Axle[1].Auto_Enable_Location[1]:=TRUE;
		 ELSIF  Auto_Data.Task_Type=2 OR Auto_Data.Task_Type=3   THEN
               Axle[0].Auto_Target_Position:=Column_Coords [Auto_Data.Start_Column] ;
			   Axle[1].Auto_Target_Position:=Layer_Coords [Auto_Data.Start_Layer]-Height_Goods_Lowered;
			   Axle[0].Auto_Enable_Location[1]:=TRUE;
			   Axle[1].Auto_Enable_Location[1]:=TRUE;
	     ELSIF  Auto_Data.Task_Type=4 THEN
			   Axle[0].Auto_Target_Position:=Column_Coords [7] ;
			   Axle[1].Auto_Target_Position:=Layer_Coords [1];
			   Axle[0].Auto_Enable_Location[1]:=TRUE;
			   Axle[1].Auto_Enable_Location[1]:=TRUE;
         END_IF;
         
		(*到达取货点*)
	    IF Axle[0].Auto_Position_Reached AND Axle[1].Auto_Position_Reached THEN
		     Axle[0].Auto_Enable_Location[1]:=FALSE;
		     Axle[1].Auto_Enable_Location[1]:=FALSE; 
	         Auto_Data.Auto_Step:=11;
	         IF Auto_Data.Task_Type=4 THEN
	         	 Auto_Data.Auto_Step:=20;
	         END_IF;
		END_IF;
		
	11:   (*伸出货叉轴准备取货*)
	    IF Auto_Data.Task_Type=1 THEN    
	    	 Master_R.LoadGoods_Apply:=1;
		     IF Station_Status[Auto_Data.Picking_Station_No].LoadGoods_Enable THEN
		 	    Axle[2].Auto_Target_Position:=Station_Coords[Auto_Data.Picking_Station_No].Z_Position;
		 	    Axle[2].Auto_Enable_Location[1]:=TRUE;
			    Stacker_R_Status_Bit.Picked_Up:=TRUE;
		    END_IF;
	    ELSIF   Auto_Data.Task_Type=2 OR Auto_Data.Task_Type=3 THEN
		       Axle[2].Auto_Target_Position:=Row_Coords[Auto_Data.Start_Row] ;
		       Axle[2].Auto_Enable_Location[1]:=TRUE; 
	    END_IF;
	    
		  IF Axle[2].Auto_Position_Reached THEN
			 Axle[2].Auto_Enable_Location[1]:=FALSE;
			 Master_R.LoadGoods_Apply:=0;
			 Auto_Data.Auto_Step:=12;
          END_IF;
		
	12:  (*抬起货叉轴*)
         Stacker_R_Status_Bit.Picked_Up:=TRUE;
	     IF Auto_Data.Task_Type=1THEN
			     Axle[1].Auto_Target_Position:= Station_Coords[Auto_Data.Picking_Station_No].Y_Position+Height_Goods_Lifted;
			     Axle[1].Auto_Enable_Location[1]:=TRUE;
		 ELSIF  Auto_Data.Task_Type=2 OR Auto_Data.Task_Type=3 THEN
			     Axle[1].Auto_Target_Position:=Layer_Coords[Auto_Data.Start_Layer] +Height_Goods_Lifted;
			     Axle[1].Auto_Enable_Location[1]:=TRUE;
		 END_IF;
			
		 IF Axle[1].Auto_Position_Reached THEN
			Axle[1].Auto_Enable_Location[1]:=FALSE;
			Auto_Data.Auto_Step:=13;
		 END_IF;
	
	13:  (*缩回货叉轴*)
	        Stacker_R_Status_Bit.Picked_Up:=TRUE;
	        Axle[2].Auto_Target_Position:= 0.0;
		    Axle[2].Auto_Enable_Location[1]:=TRUE;

		    IF Axle[2].Auto_Position_Reached THEN
			  Axle[2].Auto_Enable_Location[1]:=FALSE;
		      Auto_Data.Auto_Step:=14;
		   END_IF;
		
	14:   (*Fork_取料完成*)
             Stacker_R_Status_Bit.Picked_Up:=FALSE;
			IF Platform_Goods_Detection THEN
			    Fork_Load_Done:=TRUE;
			   Auto_Data.Auto_Step:=15;
			ELSE
				Alarm_record[2]:=TRUE;
				Auto_Data.Error_Code:=2;
			END_IF;
		
	15:  (*Fork_前往放货点*)
	      IF Auto_Data.Task_Type=1 OR Auto_Data.Task_Type=3 THEN
				Axle[0].Auto_Target_Position:=Column_Coords [Auto_Data.End_Column] ;
			    Axle[1].Auto_Target_Position:=Layer_Coords [Auto_Data.End_Layer]+Height_Goods_Lifted;
		  ELSIF Auto_Data.Task_Type=2 THEN
				Axle[0].Auto_Target_Position:=Station_Coords[Auto_Data.Placing_Station_No].X_Position;
				Axle[1].Auto_Target_Position:=Station_Coords[Auto_Data.Placing_Station_No].Y_Position+Height_Goods_Lifted;
		  END_IF;
			   Axle[0].Auto_Enable_Location[1]:=TRUE;
			   Axle[1].Auto_Enable_Location[1]:=TRUE;

		 IF Axle[0].Auto_Position_Reached AND Axle[1].Auto_Position_Reached THEN
			 Axle[0].Auto_Enable_Location[1]:=FALSE;
			 Axle[1].Auto_Enable_Location[1]:=FALSE; 
			 Auto_Data.Auto_Step:=16;
		 END_IF;
		 
	16:  (*伸出货叉轴*)
	     IF Auto_Data.Task_Type=2 THEN   
	     	  Master_R.UnLoadGoods_Apply:=1;
		     IF Station_Status[Auto_Data.Placing_Station_No].UnLoadGoods_Enable AND Fork_Goods_Detection[1]=FALSE THEN
			     Axle[2].Auto_Target_Position:=Station_Coords[Auto_Data.Placing_Station_No].Z_Position;
		     	 Axle[2].Auto_Enable_Location[1]:=TRUE;
			     Stacker_R_Status_Bit.Releasing_Goods:=TRUE;
		    END_IF;
		 ELSIF   (Auto_Data.Task_Type=1 OR Auto_Data.Task_Type=3) AND 
			((Fork_Goods_Detection[0] =FALSE AND Auto_Data.End_Row=1) OR (Fork_Goods_Detection[1]=FALSE AND Auto_Data.End_Row=2)) THEN
		    Axle[2].Auto_Target_Position:=Row_Coords[Auto_Data.End_Row];
		    Axle[2].Auto_Enable_Location[1]:=TRUE;
		    
		ELSIF  (Auto_Data.Task_Type=1 OR Auto_Data.Task_Type=3) AND Axle[2].Auto_Enable_Location[1]=FALSE AND 
		   ((Fork_Goods_Detection[0] =TRUE AND Auto_Data.End_Row=1) OR (Fork_Goods_Detection[1]=TRUE AND Auto_Data.End_Row=2))THEN
			Alarm_record[3]:=TRUE;
			Auto_Data.Error_Code:=3;
		 END_IF;
		 
		  IF Axle[2].Auto_Position_Reached THEN
			 Axle[2].Auto_Enable_Location[1]:=FALSE;
			 Master_R.UnLoadGoods_Apply:=0;
		     Auto_Data.Auto_Step:=17;
		  END_IF;
		  
	17: (*下降货叉轴*)
	        Stacker_R_Status_Bit.Releasing_Goods:=TRUE;
		     IF Auto_Data.Task_Type=2 THEN
			    Axle[1].Auto_Target_Position:= Station_Coords[Auto_Data.Placing_Station_No].Y_Position-Height_Goods_Lowered;
			    Axle[1].Auto_Enable_Location[1]:=TRUE;
		     ELSIF Auto_Data.Task_Type=1 OR Auto_Data.Task_Type=3 THEN
			    Axle[1].Auto_Target_Position:=Layer_Coords[Auto_Data.End_Layer] -Height_Goods_Lowered;
			    Axle[1].Auto_Enable_Location[1]:=TRUE;
		     END_IF;

		    IF Axle[1].Auto_Position_Reached THEN
			      Axle[1].Auto_Enable_Location[1]:=FALSE;
		          Auto_Data.Auto_Step:=18;
	        END_IF;
	
	18: (*缩回货叉轴*)
	         Stacker_R_Status_Bit.Releasing_Goods:=TRUE;
		     Axle[2].Auto_Target_Position:= 0.0;
		     Axle[2].Auto_Enable_Location[1]:=TRUE;
		     
		     IF Axle[2].Auto_Position_Reached THEN
			      Axle[2].Auto_Enable_Location[1]:=FALSE;
		          Auto_Data.Auto_Step:=19;
		     END_IF;
		  
	19:   (*Fork_放料完成*)
			 Stacker_R_Status_Bit.Releasing_Goods:=FALSE;
			 IF Platform_Goods_Detection=FALSE THEN
			      Fork_Unload_Done:=TRUE;
			      Auto_Data.Auto_Step:=20;
			 ELSE
			 	Alarm_record[4]:=TRUE;
			 	Auto_Data.Error_Code:=4;
			 END_IF;
			
	20:  (*任务完成判断*)
			Alone.Picking_Station_No:=0;
			Alone.Placing_Station_No:=0;
			Alone.Task_Type:=0;
			Alone.Start_Row:=0;
			Alone.Start_Column:=0;
			Alone.Start_Layer:=0;
			Alone.End_Row:=0;
			Alone.End_Column:=0;
			Alone.End_Layer:=0;
			Auto_Data.Task_Status:=5;
			Auto_Data.Auto_Step:=0;
			Auto_Run := FALSE;
			Record.Auto_Step:=0	;
	END_CASE; 
END_IF;
END_PROGRAM

PROGRAM 07_Manua
VAR
  AO1 : INT;
END_VAR
(*电机 位置/速度 计算
//X轴 电机每转位移数 78.54MM   减速比 10    最大运行速度M/MIN 137  加减速度0.4M/S2
//Y轴 电机每转位移数 33.35MM    减速比 39   最大运行速度M/MIN 30   加减速度0.4M/S2
//Z轴 电机每转位移数 18.43MM    减速比 15      最大运行速度M/MIN 60   加减速度0.5M/S2
//X轴  //最大速度2000MM/S
//Y轴  //最大速度500MM/S   ---1000
//Z轴  //最大速度1000MM/S----550*)

(*当前电机位置换算MM*)
Axle_attribute[0].Motor_Actual_Position:=Axle[0].o_wdCurrentPosition_F / 10.0;
Auto_Data.X_Current_Actual_Position:=Axle_attribute[0].Motor_Actual_Position - Parameter_Set.X_OffsetPos;

Axle_attribute[1].Motor_Actual_Position:=Axle[1].o_wdCurrentPosition_F / 10.0;
Auto_Data.Y_Current_Actual_Position:=Axle_attribute[1].Motor_Actual_Position -  Parameter_Set.Y_OffsetPos;

Axle_attribute[2].Motor_Actual_Position:=Axle[2].o_wdCurrentPosition_F / 10.0;
Auto_Data.Z_Current_Actual_Position:=Axle_attribute[2].Motor_Actual_Position -  Parameter_Set.Z_OffsetPos;

(*当前速度换算MM/S*)
FLT(1,Axle_X_Sew_Read.Actual_Speed ,Axle[0].o_wdCurrentSpeed_F );
FLT(1,Axle_Y_Sew_Read.Actual_Speed ,Axle[1].o_wdCurrentSpeed_F );
FLT(1,Axle_Z_Sew_Read.Actual_Speed, Axle[2].o_wdCurrentSpeed_F );
Auto_Data.X_Current_Actual_Speed:=Axle[0].o_wdCurrentSpeed_F / 1.0;
Auto_Data.Y_Current_Actual_Speed :=Axle[1].o_wdCurrentSpeed_F / 1.0;
Auto_Data.Z_Current_Actual_Speed :=Axle[2].o_wdCurrentSpeed_F / 1.0;

(*非手动模式*)
IF Mode<>2 THEN
	Axle[0].Auto_Enable_Location[2]:=FALSE;
	Axle[1].Auto_Enable_Location[2]:=FALSE;
	Axle[2].Auto_Enable_Location[2]:=FALSE;
END_IF;

(*手动控制 定位数据切换*)
IF Stacker_R_Status_Bit.Stacker_A01ManualControl THEN
	FLT(1,Master_W.X_Locate_Position,Manual.X_ManualPosition_Assist);
	FLT(1,Master_W.Y_Locate_Position,Manual.Y_ManualPosition_Assist);
	FLT(1,Master_W.Z_Locate_Position,Manual.Z_ManualPosition_Assist);
	Manual.X_Manual_Column_Assist:=Master_W.X_Locate_Column;
	Manual.Y_Manual_Layer_Assist:=Master_W.Y_Locate_Layer;
ELSE
	Manual.X_ManualPosition_Assist:=Manual.X_ManualPosition;
	Manual.Y_ManualPosition_Assist:=Manual.Y_ManualPosition;
	Manual.Z_ManualPosition_Assist:=Manual. Z_ManualPosition;
	Manual.X_Manual_Column_Assist:=Manual.X_Manual_Column_Assist;
	Manual.Y_Manual_Layer_Assist:=Manual.Y_Manual_Layer_Assist;
END_IF;

(*X轴单独控制*)
IF Mode=2 AND Manual.X_ManualStart_Position AND Fork_Middle_Detection  THEN
	IF Manual.Position_Coords_Switch = FALSE THEN
        Axle[0].Auto_Target_Position := Manual.X_ManualPosition_Assist;
	ELSE
        Axle[0].Auto_Target_Position := Column_Coords[Manual.X_Manual_Column_Assist];
    END_IF;
    Axle[0].Auto_Enable_Location[2]:=TRUE;
    Axle_X_Sew_Write.Rated_Speed:=Parameter_Set.X_Auto_Speed;
END_IF;

(* Y轴单独控制*)
IF Mode=2 AND Manual.Y_ManualStart_Position AND Fork_Middle_Detection THEN 
	IF Manual.Position_Coords_Switch = FALSE THEN
        Axle[1].Auto_Target_Position := Manual.Y_ManualPosition_Assist;
	ELSE
		Axle[1].Auto_Target_Position := Layer_Coords[Manual.Y_Manual_Layer_Assist];
    END_IF;
    Axle[1].Auto_Enable_Location[2]:=TRUE;
    Axle_Y_Sew_Write.Rated_Speed:=Parameter_Set.Y_Auto_Speed;
END_IF;

(* Z轴单独控制*)
IF Mode=2 AND Manual.Z_ManualStart_Position THEN
    Axle[2].Auto_Target_Position := Manual.Z_ManualPosition_Assist;
    Axle[2].Auto_Enable_Location[2]:=TRUE;
    Axle_Z_Sew_Write.Rated_Speed:=Parameter_Set.Z_Auto_Speed;
END_IF;

(*自动数据位置转换下发*)
Axle[0].i_wdTargetPosition_F:=(Axle[0].Auto_Target_Position + Parameter_Set.X_OffsetPos) *10.0;
Axle[1].i_wdTargetPosition_F:=(Axle[1].Auto_Target_Position + Parameter_Set.Y_OffsetPos) *10.0;
Axle[2].i_wdTargetPosition_F:=(Axle[2].Auto_Target_Position + Parameter_Set.Z_OffsetPos) *10.0;

(*定位允许*)
     (*X*)
	IF Parameter_Set.X_LimitPos>= Axle[0].Auto_Target_Position    AND 
		Parameter_Set.X_NegativePos<= Axle[0].Auto_Target_Position    AND Fork_Middle_Detection THEN
	    Positioning_Enable[0] :=TRUE;
	ELSE
		Positioning_Enable[0] :=FALSE;
	END_IF;
	(*Y*)
	IF Parameter_Set.Y_LimitPos>= Axle[1].Auto_Target_Position    AND 
		Parameter_Set.Y_NegativePos<= Axle[1].Auto_Target_Position   THEN
	    Positioning_Enable[1] :=TRUE;
	ELSE
		Positioning_Enable[1] :=FALSE;
	END_IF;
	(*Z*)
	IF Parameter_Set.Z_LimitPos>=Axle[2].Auto_Target_Position    AND 
		Parameter_Set.Z_NegativePos<=Axle[2].Auto_Target_Position THEN
	    Positioning_Enable[2] :=TRUE;
	ELSE
		Positioning_Enable[2] :=FALSE;
	END_IF;
(*开始定位*)
IF ( Axle[0].Auto_Enable_Location[1] OR Axle[0].Auto_Enable_Location[2] ) AND Positioning_Enable[0] THEN
	Axle_X_Sew_Control_Bit.Ramp_Bus_StartStop:=TRUE;
	Axle_X_Sew_Control_Bit.Enable_Application_Stop:=TRUE;
	Axle_X_Sew_Write.Set_Mode:=400;
ELSE
	Axle_X_Sew_Control_Bit.Ramp_Bus_StartStop:=FALSE;
END_IF;

IF  ( Axle[1].Auto_Enable_Location[1] OR Axle[1].Auto_Enable_Location[2]  ) AND Positioning_Enable[1] THEN
	Axle_Y_Sew_Control_Bit.Ramp_Bus_StartStop:=TRUE;
	Axle_Y_Sew_Control_Bit.Enable_Application_Stop:=TRUE;
	Axle_Y_Sew_Write.Set_Mode:=400;
ELSE
	Axle_Y_Sew_Control_Bit.Ramp_Bus_StartStop:=FALSE;
END_IF;

IF  ( Axle[2].Auto_Enable_Location[1] OR Axle[2].Auto_Enable_Location[2]  ) AND Positioning_Enable[2] THEN
	Axle_Z_Sew_Control_Bit.Ramp_Bus_StartStop:=TRUE;
	Axle_Z_Sew_Control_Bit.Enable_Application_Stop:=TRUE;
	Axle_Z_Sew_Write.Set_Mode:=400;
ELSE
	Axle_Z_Sew_Control_Bit.Ramp_Bus_StartStop:=FALSE;
END_IF;

(*自动速度及模式设置MM/S*)
Parameter_Set.Y_LoadGoods_Speed:=50;
	(*X*)
	IF DInput.Walk_Deceleration AND Axle_X_Sew_Control_Bit.Ramp_Bus_StartStop THEN
		Axle_X_Sew_Write.Rated_Speed:=500;
	ELSIF Axle_X_Sew_Control_Bit.Ramp_Bus_StartStop THEN
	Axle_X_Sew_Write.Rated_Speed:=Parameter_Set.X_Auto_Speed;
	END_IF;
	(*Y*)
	IF Auto_Data.Auto_Step=12 OR Auto_Data.Auto_Step=17  THEN
		Axle_Y_Sew_Write.Rated_Speed:=Parameter_Set.Y_LoadGoods_Speed;
	ELSIF Axle_Y_Sew_Control_Bit.Ramp_Bus_StartStop THEN
		IF DInput.Lift_Deceleration  THEN
			 Axle_Y_Sew_Write.Rated_Speed:=300;
		ELSE
	   Axle_Y_Sew_Write.Rated_Speed:=Parameter_Set.Y_Auto_Speed;
	   END_IF;
	END_IF;
	(*Z*)
	IF  Axle_Z_Sew_Control_Bit.Ramp_Bus_StartStop THEN
	Axle_Z_Sew_Write.Rated_Speed:=Parameter_Set.Z_Auto_Speed;
	END_IF;
	
(*加减速度设置*)
IF  Axle_X_Sew_Control_Bit.Ramp_Bus_StartStop THEN
Axle_X_Sew_Write.Acceleration:=Parameter_Set.X_Acceleration;
Axle_X_Sew_Write.Deceleration:=Parameter_Set.X_Deceleration;
END_IF;

IF  Axle_Y_Sew_Control_Bit.Ramp_Bus_StartStop THEN
Axle_Y_Sew_Write.Acceleration:=Parameter_Set.Y_Acceleration;
Axle_Y_Sew_Write.Deceleration:=Parameter_Set.Y_Deceleration;
END_IF;

IF  Axle_Z_Sew_Control_Bit.Ramp_Bus_StartStop THEN
Axle_Z_Sew_Write.Acceleration:=Parameter_Set.Z_Acceleration;
Axle_Z_Sew_Write.Deceleration:=Parameter_Set.Z_Deceleration;
END_IF;

(*励磁*)
IF E_Stop =FALSE THEN
	Axle_X_Sew_Control_Bit.Enable_Emergency_Stop:=TRUE;
	Axle_Y_Sew_Control_Bit.Enable_Emergency_Stop:=TRUE;
	Axle_Z_Sew_Control_Bit.Enable_Emergency_Stop:=TRUE;
ELSE
	Axle_X_Sew_Control_Bit.Enable_Emergency_Stop:=FALSE;
	Axle_X_Sew_Control_Bit.Enable_Application_Stop:=FALSE;
	Axle_Y_Sew_Control_Bit.Enable_Emergency_Stop:=FALSE;
	Axle_Y_Sew_Control_Bit.Enable_Application_Stop:=FALSE;
	Axle_Z_Sew_Control_Bit.Enable_Emergency_Stop:=FALSE;
	Axle_Z_Sew_Control_Bit.Enable_Application_Stop:=FALSE;
END_IF;

(*软硬限位  正反转允许判断*)
     (*X*)
	IF Parameter_Set.X_LimitPos>Auto_Data.X_Current_Actual_Position AND DInput.Walk_Forward_TO_Pos=FALSE  AND DInput.Walk_INV_Power  AND 
		Fork_Middle_Detection AND (DInput.Forward_Laser_Stop OR HMI.Laser_Close ) AND TS0 THEN
	    Axle[0].Forward_Enable:=TRUE;
	ELSE
		Axle[0].Forward_Enable:=FALSE;
	END_IF;
	IF Parameter_Set.X_NegativePos<Auto_Data.X_Current_Actual_Position AND DInput.Walk_Reverse_TO_Pos=FALSE   AND DInput.Walk_INV_Power  AND 
		Fork_Middle_Detection AND (DInput.Reverse_Laser_Stop OR HMI.Laser_Close ) AND TS0 THEN
	    Axle[0].Reverse_Enable:=TRUE;
	ELSE
		Axle[0].Reverse_Enable:=FALSE;
	END_IF;
	(*Y*)
	IF Parameter_Set.Y_LimitPos>Auto_Data.Y_Current_Actual_Position AND DInput.Lift_Up_TO_Pos=FALSE  AND DInput.Lift_INV_Power   AND (Fork_Middle_Detection OR Manual_Y_Force_Enable) AND TS0 THEN
	    Axle[1].Forward_Enable:=TRUE;
	ELSE
		Axle[1].Forward_Enable:=FALSE;
	END_IF;
	IF Parameter_Set.Y_NegativePos<Auto_Data.Y_Current_Actual_Position AND DInput.Lift_Down_TO_Pos=FALSE  AND DInput.Lift_INV_Power   AND (Fork_Middle_Detection OR Manual_Y_Force_Enable) AND TS0 THEN
	    Axle[1].Reverse_Enable:=TRUE;
	ELSE
		Axle[1].Reverse_Enable:=FALSE;
	END_IF;
	(*Z*)
	IF Parameter_Set.Z_LimitPos>Auto_Data.Z_Current_Actual_Position AND DInput.Fork_Left_To_Pos=FALSE  AND DInput.Fork_INV_Power AND TS0 THEN
	    Axle[2].Forward_Enable:=TRUE;
	ELSE
		Axle[2].Forward_Enable:=FALSE;
	END_IF;
	IF Parameter_Set.Z_NegativePos<Auto_Data.Z_Current_Actual_Position AND DInput.Fork_Right_To_Pos=FALSE  AND DInput.Fork_INV_Power AND TS0 THEN
	    Axle[2].Reverse_Enable:=TRUE;
	ELSE
		Axle[2].Reverse_Enable:=FALSE;
	END_IF;
(*手动模式*)
IF Mode=2 THEN
	    Axle_X_Sew_Control_Bit.Forward_Jog:=Axle[0].Jog_Forward AND Axle[0].Forward_Enable ;
		Axle_X_Sew_Control_Bit.Reverse_Jog:=Axle[0].Jog_Reverse AND Axle[0].Reverse_Enable;
		Axle_Y_Sew_Control_Bit.Forward_Jog:=Axle[1].Jog_Forward AND Axle[1].Forward_Enable;
		Axle_Y_Sew_Control_Bit.Reverse_Jog:=Axle[1].Jog_Reverse AND Axle[1].Reverse_Enable;
		Axle_Z_Sew_Control_Bit.Forward_Jog:=Axle[2].Jog_Forward AND Axle[2].Forward_Enable;
		Axle_Z_Sew_Control_Bit.Reverse_Jog:=Axle[2].Jog_Reverse AND Axle[2].Reverse_Enable;
		
		IF Axle_X_Sew_Control_Bit.Forward_Jog OR Axle_X_Sew_Control_Bit.Reverse_Jog THEN
			Axle_X_Sew_Write.Set_Mode:=100;
			Axle_X_Sew_Control_Bit.Enable_Application_Stop:=TRUE;
			Axle_X_Sew_Write.Rated_Speed:=Parameter_Set.X_Manual_Speed;
			Axle_X_Sew_Write.Acceleration:=50;
            Axle_X_Sew_Write.Deceleration:=50;
		END_IF;
		IF Axle_Y_Sew_Control_Bit.Forward_Jog OR  Axle_Y_Sew_Control_Bit.Reverse_Jog THEN
			Axle_Y_Sew_Write.Set_Mode:=101;
			Axle_Y_Sew_Control_Bit.Enable_Application_Stop:=TRUE;
			Axle_Y_Sew_Write.Rated_Speed:=Parameter_Set.Y_Manual_Speed;
			Axle_Y_Sew_Write.Acceleration:=50;
            Axle_Y_Sew_Write.Deceleration:=50;
		END_IF;
		IF Axle_Z_Sew_Control_Bit.Forward_Jog OR Axle_Z_Sew_Control_Bit.Reverse_Jog THEN
			Axle_Z_Sew_Write.Set_Mode:=100;
			Axle_Z_Sew_Control_Bit.Enable_Application_Stop:=TRUE;
			Axle_Z_Sew_Write.Rated_Speed:=Parameter_Set.Z_Manual_Speed;
			Axle_Z_Sew_Write.Acceleration:=50;
            Axle_Z_Sew_Write.Deceleration:=50;
		END_IF;
END_IF;

(*定位位置到达判断*)
Axle_attribute[0].Position_Difference:=ABS(Auto_Data.X_Current_Actual_Position  - Axle[0].Auto_Target_Position);
Axle_attribute[1].Position_Difference:=ABS(Auto_Data.Y_Current_Actual_Position  - Axle[1].Auto_Target_Position);
Axle_attribute[2].Position_Difference:=ABS(Auto_Data.Z_Current_Actual_Position  - Axle[2].Auto_Target_Position);
AO1:=0;
FOR AO1:=0 TO 2 DO
    IF Axle_attribute[AO1].Position_Difference< 2.0 THEN
         Axle_attribute[AO1].Position_Reached := TRUE;
    ELSE
         Axle_attribute[AO1].Position_Reached:= FALSE;
	END_IF;
END_FOR;
Axle[0].Auto_Position_Reached:=Axle_attribute[0].Position_Reached AND  Axle_X_Sew_Status_Bit.Position_Arrive AND  ( Axle[0].Auto_Enable_Location[1] OR Axle[0].Auto_Enable_Location[2] ) ;
Axle[1].Auto_Position_Reached:=Axle_attribute[1].Position_Reached AND  Axle_Y_Sew_Status_Bit.Position_Arrive AND  ( Axle[1].Auto_Enable_Location[1] OR Axle[1].Auto_Enable_Location[2] ) ;
Axle[2].Auto_Position_Reached:=Axle_attribute[2].Position_Reached AND  Axle_Z_Sew_Status_Bit.Position_Arrive  AND  ( Axle[2].Auto_Enable_Location[1] OR Axle[2].Auto_Enable_Location[2] ) ;

(*复位手动定位*)
IF (Axle_X_Sew_Status_Bit.Position_Arrive AND Axle_X_Sew_Control_Bit.Ramp_Bus_StartStop  AND Axle[0].Auto_Position_Reached )OR Auto_Data.Error_Code<>0 THEN
	Axle[0].Auto_Enable_Location[2]:=FALSE;
END_IF;
IF (Axle_Y_Sew_Status_Bit.Position_Arrive AND Axle_Y_Sew_Control_Bit.Ramp_Bus_StartStop  AND Axle[1].Auto_Position_Reached )OR Auto_Data.Error_Code<>0 THEN
	Axle[1].Auto_Enable_Location[2]:=FALSE;
END_IF;
IF (Axle_Z_Sew_Status_Bit.Position_Arrive AND Axle_Z_Sew_Control_Bit.Ramp_Bus_StartStop  AND Axle[2].Auto_Position_Reached )OR Auto_Data.Error_Code<>0 THEN
	Axle[2].Auto_Enable_Location[2]:=FALSE;
END_IF;

(*复位Sew_Control_Bit.使能应用停止*)
OUT_T(Axle_X_Sew_Control_Bit.Forward_Jog=FALSE AND Axle_X_Sew_Control_Bit.Reverse_Jog=FALSE AND Axle[0].Auto_Enable_Location[1]=FALSE AND Axle[0].Auto_Enable_Location[2]=FALSE AND Axle_X_Sew_Control_Bit.Enable_Application_Stop,TC4,2);
IF   TS4 THEN
	rst(TS4,TC4);
	  Axle_X_Sew_Control_Bit.Enable_Application_Stop:=FALSE;
END_IF;
OUT_T(Axle_Y_Sew_Control_Bit.Forward_Jog=FALSE AND Axle_Y_Sew_Control_Bit.Reverse_Jog=FALSE AND Axle[1].Auto_Enable_Location[1]=FALSE AND Axle[1].Auto_Enable_Location[2]=FALSE AND  Axle_Y_Sew_Control_Bit.Enable_Application_Stop,TC5,3);
IF  TS5 THEN
	rst(TS5,TC5);
	  Axle_Y_Sew_Control_Bit.Enable_Application_Stop:=FALSE;
END_IF;
OUT_T(Axle_Z_Sew_Control_Bit.Forward_Jog=FALSE AND Axle_Z_Sew_Control_Bit.Reverse_Jog=FALSE AND Axle[2].Auto_Enable_Location[1]=FALSE AND Axle[2].Auto_Enable_Location[2]=FALSE AND Axle_Z_Sew_Control_Bit.Enable_Application_Stop,TC6,3);
IF   TS6 THEN
	rst(TS6,TC6);
	  Axle_Z_Sew_Control_Bit.Enable_Application_Stop:=FALSE;
END_IF;

(*故障及状态获取*)
IF Axle_X_Sew_Status_Bit.Error THEN
	Axle_X_Alalm := Axle_X_Sew_Read.Main_Status_Fault;
	Axle_X_Status := 0;
ELSE
	Axle_X_Alalm:=0 ;
	Axle_X_Status:=Axle_X_Sew_Read.Main_Status_Fault ;
END_IF;
IF Axle_Y_Sew_Status_Bit.Error THEN
	Axle_Y_Alalm:=Axle_Y_Sew_Read.Main_Status_Fault;
	Axle_Y_Status:=0;
ELSE
	Axle_Y_Alalm:=0;
	Axle_Y_Status:=Axle_Y_Sew_Read.Main_Status_Fault;
END_IF;

IF Axle_Z_Sew_Status_Bit.Error THEN
	Axle_Z_Alalm:=Axle_Z_Sew_Read.Main_Status_Fault;
	Axle_Z_Status:=0;
ELSE
	Axle_Z_Alalm:=0;
	Axle_Z_Status:=Axle_Z_Sew_Read.Main_Status_Fault;
END_IF;


(*Fork_在零点*)
IF Fork_Middle_Detection AND Auto_Data.Z_Current_Actual_Position>-2.0 AND Auto_Data.Z_Current_Actual_Position<2.0 THEN
	Fork_Zero:=TRUE;
ELSE
	Fork_Zero:=FALSE;
END_IF;

(*堆垛机当前位置判断*)	
Stacker_Current_Column:=0;
AO1:=0;
FOR AO1:=1 TO 14 DO
	IF Auto_Data.X_Current_Actual_Position >(Column_Coords[AO1]-50.0) AND Auto_Data.X_Current_Actual_Position <(Column_Coords[AO1]+50.0) THEN
	     Stacker_Current_Column:=AO1;
		 EXIT;
	END_IF;
END_FOR;
Stacker_Current_Layer:=0;
AO1:=0;
FOR AO1:=1 TO 5 DO
	IF Auto_Data.Y_Current_Actual_Position >(Layer_Coords[AO1]-50.0) AND Auto_Data.Y_Current_Actual_Position <(Layer_Coords[AO1]+70.0) THEN
		Stacker_Current_Layer:=AO1;
		EXIT;
	END_IF;
END_FOR;
END_PROGRAM

PROGRAM 08_Alarm
VAR
  AO1 : INT;
  AO2 : INT;
  Alarm_No : INT;
  Rising : BOOL;
END_VAR
(*错误码*)
(*急停*)
IF TS0 THEN
IF E_Stop  THEN
	Alarm_record[1]:=TRUE;
	Auto_Data.Error_Code := 1;
END_IF;

(*Fork_未取到料箱报警
Auto_Data.Error_Code:=2;*)

(*//Fork_放货时库位有料箱报警
//Auto_Data.Error_Code:=3;*)

(*//Fork_放货不成功报警
//Auto_Data.Error_Code:=4;*)


(*//地面站的数据链接状态*)
IF M340 THEN
	Alarm_record[5]:=TRUE;
	Auto_Data.Error_Code := 5;
END_IF;

(*SEW的数据链接状态_*)
IF M320 THEN
	Alarm_record[6]:=TRUE;
	Auto_Data.Error_Code := 6;
END_IF;
IF M322 THEN
	Alarm_record[7]:=TRUE;
	Auto_Data.Error_Code := 7;
END_IF;
IF M324 THEN
	Alarm_record[8]:=TRUE;
	Auto_Data.Error_Code := 8;
END_IF;

(*货叉轴 原点开关异常*)
IF Fork_Middle_Detection = FALSE AND Auto_Data.Z_Current_Actual_Position=0.0 THEN
    Alarm_record[9]:=TRUE;
    Auto_Data.Error_Code := 9;
END_IF;

(*WCS指令错误*)
IF (Wcs_interface.Task_Type < 0 OR Wcs_interface.Task_Type  > 4 OR
    Wcs_interface.Start_Row > 2 OR Wcs_interface.Start_Column > 14 OR Wcs_interface.Start_Layer > 5 OR
	Wcs_interface.End_Row > 2 OR Wcs_interface.End_Column > 14 OR Wcs_interface.End_Layer > 5 ) AND Mode<=1  THEN
    Alarm_record[10]:=TRUE;
    Auto_Data.Error_Code := 10;
END_IF;

(*上位机急停*)
IF Master_W.EStop_Control<>0 THEN 
   Auto_Data.Error_Code :=11;
   Alarm_record[11]:=TRUE;
END_IF;


IF DInput.Lift_Stall=FALSE   THEN
    Alarm_record[12]:=TRUE;
    Auto_Data.Error_Code := 12;
END_IF;

IF DInput.Lift_Rope_Loosening1=FALSE AND HMI.Overload_Detection_Close=FALSE THEN
    Alarm_record[13]:=TRUE;
    Auto_Data.Error_Code := 13;
END_IF;

IF DInput.Lift_Rope_Loosening2=FALSE AND HMI.Overload_Detection_Close=FALSE THEN
    Alarm_record[14]:=TRUE;
    Auto_Data.Error_Code := 14;
END_IF;

IF DInput.Lift_Overload1=FALSE  AND HMI.Overload_Detection_Close=FALSE THEN
    Alarm_record[15]:=TRUE;
    Auto_Data.Error_Code := 15;
END_IF;

IF DInput.Lift_Overload2=FALSE  AND HMI.Overload_Detection_Close=FALSE THEN
    Alarm_record[16]:=TRUE;
    Auto_Data.Error_Code := 16;
END_IF;

IF DInput.Air_Error  THEN
    Alarm_record[17]:=TRUE;
    Auto_Data.Error_Code := 17;
END_IF;

IF DInput.Optical_Error=FALSE THEN
     Alarm_record[18]:=TRUE;
     Auto_Data.Error_Code := 18;
END_IF;

IF Fork_Alarm.Fork_Left_collapse_Alarm1 THEN
    Alarm_record[19]:=TRUE;
    Auto_Data.Error_Code := 19;
END_IF;

IF Fork_Alarm.Fork_Left_collapse_Alarm2  THEN
    Alarm_record[20]:=TRUE;
    Auto_Data.Error_Code := 20;
END_IF;

IF Fork_Alarm.Fork_Left_Width_Alarm1  THEN
    Alarm_record[21]:=TRUE;
    Auto_Data.Error_Code := 21;
END_IF;

IF Fork_Alarm.Fork_Left_Width_Alarm2 THEN
    Alarm_record[22]:=TRUE;
    Auto_Data.Error_Code := 22;
END_IF;

IF Fork_Alarm.Fork_Left_Height_Alarm THEN
    Alarm_record[23]:=TRUE;
    Auto_Data.Error_Code := 23;
END_IF;

IF Fork_Alarm.Fork_Right_collapse_Alarm1  THEN
    Alarm_record[24]:=TRUE;
    Auto_Data.Error_Code := 24;
END_IF;

IF Fork_Alarm.Fork_Right_collapse_Alarm2 THEN
    Alarm_record[25]:=TRUE;
    Auto_Data.Error_Code := 25;
END_IF;

IF Fork_Alarm.Fork_Right_Width_Alarm1  THEN
    Alarm_record[26]:=TRUE;
    Auto_Data.Error_Code := 26;
END_IF;

IF Fork_Alarm.Fork_Right_Width_Alarm2  THEN
    Alarm_record[27]:=TRUE;
    Auto_Data.Error_Code := 27;
END_IF;

IF Fork_Alarm.Fork_Right_Height_Alarm  THEN
    Alarm_record[28]:=TRUE;
    Auto_Data.Error_Code := 28;
END_IF;

(*激光避障停止*)
IF (DInput.Forward_Laser_Stop=FALSE OR  DInput.Reverse_Laser_Stop=FALSE ) AND Mode<=2 AND HMI.Laser_Close=FALSE THEN
	Laser.Obstacle_Alarm:=TRUE;
	Alarm_record[29]:=TRUE;
	Auto_Data.Error_Code := 29;
END_IF;

IF DInput.Forward_Laser_Alarm =FALSE  THEN
    Alarm_record[30]:=TRUE;
    Auto_Data.Error_Code := 30;
END_IF;

IF DInput.Reverse_Laser_Alarm =FALSE THEN
   Alarm_record[31]:=TRUE;
   Auto_Data.Error_Code := 31;
END_IF;

(*入库任务货叉有料*)
(*Alarm_record[32]:=TRUE;
Auto_Data.错误码:=32;*)
	
IF  Axle_X_Sew_Status_Bit.Error THEN
	Alarm_record[33]:=TRUE;
	Auto_Data.Error_Code := 33;
END_IF;
IF  Axle_Y_Sew_Status_Bit.Error THEN
	Alarm_record[34]:=TRUE;
	Auto_Data.Error_Code := 34;
END_IF;
IF  Axle_Z_Sew_Status_Bit.Error THEN
	Alarm_record[35]:=TRUE;
	Auto_Data.Error_Code := 35;
END_IF;	

IF DInput.Platform_Safety_Latch1=FALSE OR DInput.Platform_Safety_Latch2=FALSE THEN 
	 Alarm_record[36]:=TRUE;
   Auto_Data.Error_Code := 36;
END_IF;
END_IF;		
		 	
(*货叉光电报警*)
IF Mode<=1 THEN
	(*左侧*)
	IF DInput.Left_collapse_Signal1 AND Fork_Middle_Detection AND Axle_Z_Sew_Control_Bit.Ramp_Bus_StartStop=FALSE THEN
		Fork_Alarm.Fork_Left_collapse_Alarm1:=TRUE;
	END_IF;
	IF DInput.Left_collapse_Signal2 AND Fork_Middle_Detection AND Axle_Z_Sew_Control_Bit.Ramp_Bus_StartStop=FALSE THEN
		Fork_Alarm.Fork_Left_collapse_Alarm2:=TRUE;
	END_IF;
		Fork_Alarm.Fork_Left_Width_Alarm1:=DInput.Left_Width_Signal1;
		Fork_Alarm.Fork_Left_Width_Alarm2:=DInput.Left_Width_Signal2;
		Fork_Alarm.Fork_Left_Height_Alarm:=DInput.Left_Height_Signal;
	(*右侧*)
	IF DInput.Right_collapse_Signal1 AND Fork_Middle_Detection  AND Axle_Z_Sew_Control_Bit.Ramp_Bus_StartStop=FALSE THEN
		Fork_Alarm.Fork_Right_collapse_Alarm1:=TRUE;
	END_IF;
	IF DInput.Right_collapse_Signal2 AND Fork_Middle_Detection AND Axle_Z_Sew_Control_Bit.Ramp_Bus_StartStop=FALSE THEN
		Fork_Alarm.Fork_Right_collapse_Alarm2:=TRUE;
	END_IF;
		Fork_Alarm.Fork_Right_Width_Alarm1:=DInput.Right_Width_Signal1 ;
		Fork_Alarm.Fork_Right_Width_Alarm2:=DInput.Right_Width_Signal2;
		Fork_Alarm.Fork_Right_Height_Alarm:=DInput.Right_Height_Signal;
END_IF;

(*报警弹窗*)
IF Auto_Data.Error_Code<> 0 AND NOT Screen_Assistance THEN
	HMI_Screen:=5;
END_IF;
Screen_Assistance:=Auto_Data.Error_Code<> 0;

(*报警记录*)
(*IF SM413 AND NOT Rising THEN
AO1:=0;
     FOR AO1:=AO2 TO 40 DO
            IF Alarm_record[AO1] AND  (Alarm_No<>AO1 OR AO2=0) THEN
                 Alarm_No:= AO1;
                 AO2:=AO1;
    	         EXIT;
            END_IF;
            IF AO1=40 AND AO2=0 THEN
            	Alarm_No:=0;
            END_IF;
          IF AO1=40 THEN
    	      AO2:=0;
         END_IF;
    END_FOR;
END_IF;
Auto_Data.Error_Code:= Alarm_No;
Rising :=SM413 ;*)

(*报警复位*)
IF (HMI.Alarm_Reset OR DInput.Alarm_Reset OR Master_W.Reset_Control=1) AND  Auto_Data.Error_Code<>0 THEN
     K4M800:=0;
     K4M816:=0;
     K4M832:=0;
    Auto_Data.Error_Code := 0;
	(*Auto_Data.Task_Status:=0;*)
	Axle[0].Auto_Enable_Location[1]:=FALSE;
	Axle[1].Auto_Enable_Location[1]:=FALSE;
	Axle[2].Auto_Enable_Location[1]:=FALSE;
	Axle[0].Auto_Enable_Location[2]:=FALSE;
	Axle[1].Auto_Enable_Location[2]:=FALSE;
	Axle[2].Auto_Enable_Location[2]:=FALSE;
    Auto_Data.Auto_Step := 0;
    Auto_Run := FALSE;
    Laser.Obstacle_Alarm:=FALSE;
    Axle_X_Sew_Control_Bit.Alarm_Reset:=TRUE;
    Axle_Y_Sew_Control_Bit.Alarm_Reset:=TRUE;
    Axle_Z_Sew_Control_Bit.Alarm_Reset:=TRUE;
    Fork_Alarm.Fork_Left_collapse_Alarm1:=FALSE;
    Fork_Alarm.Fork_Left_collapse_Alarm2:=FALSE;
    Fork_Alarm.Fork_Right_collapse_Alarm1:=FALSE;
    Fork_Alarm.Fork_Right_collapse_Alarm2:=FALSE;
    Fork_Alarm.Fork_Left_Width_Alarm1:=FALSE;
	Fork_Alarm.Fork_Left_Width_Alarm2:=FALSE;
    Fork_Alarm.Fork_Left_Height_Alarm:=FALSE;
    Fork_Alarm.Fork_Right_Width_Alarm1:=FALSE ;
	Fork_Alarm.Fork_Right_Width_Alarm2:=FALSE;
	Fork_Alarm.Fork_Right_Height_Alarm:=FALSE;
    Resetting_Alarm := TRUE;
ELSE
    Resetting_Alarm := FALSE;
     Axle_X_Sew_Control_Bit.Alarm_Reset:=FALSE;
     Axle_Y_Sew_Control_Bit.Alarm_Reset:=FALSE;
     Axle_Z_Sew_Control_Bit.Alarm_Reset:=FALSE;
END_IF;
  
  (*警告码*)  	
  Warning_Code:=0;
IF Parameter_Set.X_LimitPos< Axle[0].Auto_Target_Position OR Parameter_Set.X_NegativePos> Axle[0].Auto_Target_Position   THEN
	Warning_Code:=1;
END_IF;
IF Parameter_Set.Y_LimitPos<Axle[1].Auto_Target_Position  OR Parameter_Set.Y_NegativePos> Axle[1].Auto_Target_Position   THEN
	Warning_Code:=2;
END_IF;
IF Parameter_Set.Z_LimitPos<Axle[2].Auto_Target_Position  OR Parameter_Set.Z_NegativePos>Axle[2].Auto_Target_Position THEN
	Warning_Code:=3;
END_IF;
IF DInput.Forward_Laser_Stop=FALSE  THEN
	Warning_Code:=4;
END_IF;
IF DInput.Reverse_Laser_Stop=FALSE  THEN
	Warning_Code:=5;
END_IF;
IF Parameter_Set.X_LimitPos<Auto_Data.X_Current_Actual_Position OR DInput.Walk_Forward_TO_Pos THEN
	Warning_Code:=6;
END_IF;
IF Parameter_Set.X_NegativePos>Auto_Data.X_Current_Actual_Position OR DInput.Walk_Reverse_TO_Pos THEN
	Warning_Code:=7;
END_IF;
IF Parameter_Set.Y_LimitPos<Auto_Data.Y_Current_Actual_Position OR DInput.Lift_Up_TO_Pos THEN
	Warning_Code:=8;
END_IF;
IF Parameter_Set.Y_NegativePos>Auto_Data.Y_Current_Actual_Position AND DInput.Lift_Down_TO_Pos THEN
	Warning_Code:=9;
END_IF;
IF Parameter_Set.Z_LimitPos<Auto_Data.Z_Current_Actual_Position OR DInput.Fork_Left_To_Pos THEN
	Warning_Code:=10;
END_IF;
IF Parameter_Set.Z_NegativePos>Auto_Data.Z_Current_Actual_Position OR DInput.Fork_Right_To_Pos THEN
	Warning_Code:=11;
END_IF;
END_PROGRAM

PROGRAM 03_Func
(*急停*)
 IF E_Stop=FALSE AND Laser.Obstacle_Alarm=FALSE AND Auto_Data.Error_Code=0 AND Master_W.EStop_Control=0 THEN
 	DOutput.Walk_INV_Stop:=TRUE;
 	DOutput.Fork_INV_Stop:=TRUE;
 ELSE
 	DOutput.Walk_INV_Stop:=FALSE;
 	DOutput.Fork_INV_Stop:=FALSE;
 END_IF;
(*实际扭矩.150停机 *)
 OUT_T((ABS(Axle_Y_Sew_Read.Actual_Torque)>1500 ),TC7,20);
  IF E_Stop=FALSE AND TS7=FALSE AND Auto_Data.Error_Code=0  AND Master_W.EStop_Control=0 THEN
 	DOutput.Lift_INV_Stop:=TRUE;
 ELSE
 	DOutput.Lift_INV_Stop:=FALSE;
 END_IF;

(*SM411~SM414‌：分别10ms、100ms、1s、1min的时钟脉冲信号*)
(*堆垛机静止中*)
IF Auto_Data.Auto_Step=0 THEN
	Stacker_Stationary :=TRUE;
ELSE
	Stacker_Stationary :=FALSE;
END_IF;

(*Mode_ 0联机 1单机 2手动 3维修*)
IF  DInput.Maintain_Run=FALSE  THEN
	Mode:=3;
ELSE
	(*主站切换模式*)
	IF Master_W.Mode_Switch<>Mode_Record AND Stacker_Stationary THEN
		Mode_Record :=Master_W.Mode_Switch;
		Mode:=Master_W.Mode_Switch;
	END_IF;

   (*HMI切换模式*)
	IF HMI.OnLine_Mode_Switch AND Stacker_Stationary THEN
		Mode:=0;
		ELSIF HMI.Single_Mode_Switch AND Stacker_Stationary THEN
		Mode:=1;
		ELSIF HMI.Manual_Mode_Switch AND Stacker_Stationary THEN
		Mode:=2;
	END_IF;
END_IF;

Maintenance_Mode_Stop:=DInput.Maintain_Run;

(*运行开关打开后默认切换手动模式*)
IF DInput.Maintain_Run AND NOT Maintenance_Mode_Stop THEN
	Mode:=2;
END_IF;
(*Maintenance_Mode_Stop:=DInput.Maintain_Run;*)

(*模式显示*)
OnLine_Mode:=Mode=0;
Single_Mode:=Mode=1;
Manual_Mode:=Mode=2;
Maintenance_Mode:=Mode=3;

(*语言切换*)
IF Language>3 OR Language=0 THEN
	Language:=1;
END_IF;
INCP(Language_Switch,Language);

(*密码权限-管理者*)
IF DInput.Admin=FALSE THEN
	Password:=0;
	DOutput.Buzzer:=FALSE;
	HMI.Laser_Close:=FALSE;
ELSE
	DOutput.Buzzer:=TRUE;
END_IF;
	
(*任务类型显示*)
HMI.Single_RK_Type:=Alone.Task_Type=1;
HMI.Single_CK_Type:=Alone.Task_Type=2;
HMI.Single_YK_Type:=Alone.Task_Type=3;
HMI.OnLine_RK_Type:=Wcs_interface.Task_Type=1;
HMI.OnLine_CK_Type:=Wcs_interface.Task_Type=2;
HMI.OnLine_YK_Type:=Wcs_interface.Task_Type=3;
HMI.Auto_RK_Type:=Auto_Data.Task_Type=1;
HMI.Auto_CK_Type:=Auto_Data.Task_Type=2;
HMI.Auto_YK_Type:=Auto_Data.Task_Type=3;
	
(*雷达区域切换*)
IF Auto_Data.X_Current_Actual_Position >24000.0 THEN
		DOutput.Walk_Forward_Laser_Mode1:=TRUE;
ELSE
		DOutput.Walk_Forward_Laser_Mode1:=FALSE;
END_IF;

IF Auto_Data.X_Current_Actual_Position <300.0 THEN
		DOutput.Walk_Reverse_Laser_Mode1:=TRUE;
ELSE
		DOutput.Walk_Reverse_Laser_Mode1:=FALSE;
END_IF;
END_PROGRAM

PROGRAM 09_Drive
(*数据提取*)
BMOV (1,U0\G4096,8, D100);
BMOV(1, D130,8, U0\G12288);

BMOV (1,U0\G4112,8, D110 );
BMOV (1,D140,8, U0\G12304 );

BMOV(1, U0\G4128,8, D120 );
BMOV(1, D150,8, U0\G12320 );

(*数据拆解*)
MOV (1, D100, K4M200);
MOV (1, D110, K4M220);
MOV (1, D120, K4M240);

MOV (1,K4M260 , D130);
MOV (1,K4M280 , D140);
MOV (1,K4M300 , D150);

(*通讯状态*)
MOV (1,U0\G3104, K4M320);
END_PROGRAM

PROGRAM 04Master
(*数据提取*)
BMOV (1, U2\G4096 ,30,D3000 );
BMOV (1,D3050 ,30,U2\G12288 );

MOV (1, D3024 ,K4M2500);
MOV (1,K4M2000 ,D3078 );

(*通讯状态*)
MOV (1,U2\G3104 ,K4M340);

(*Write*)
Wcs_interface.Task_ID:=Master_W.Task_ID;
Wcs_interface.Task_Type:=Master_W.Task_Type;
Wcs_interface.Picking_Station_No:=Master_W.Picking_Station_No;
Wcs_interface.Placing_Station_No:=Master_W.Placing_Station_No;
Wcs_interface.Start_Row:=Master_W.Start_Row;
Wcs_interface.Start_Column:=Master_W.Start_Column;
Wcs_interface.Start_Layer:=Master_W.Start_Layer;
Wcs_interface.End_Row:=Master_W.End_Row;
Wcs_interface.End_Column:=Master_W.End_Column;
Wcs_interface.End_Layer:=Master_W.End_Layer;
IF Master_W.LoadGoods_Enable_B1=1 THEN
	Station_Status[1].LoadGoods_Enable:=TRUE;
ELSE
	Station_Status[1].LoadGoods_Enable:=FALSE;
END_IF;
IF Master_W.LoadGoods_Enable_B2=1 THEN
	Station_Status[2].LoadGoods_Enable:=TRUE;
ELSE
	Station_Status[2].LoadGoods_Enable:=FALSE;
END_IF;
IF Master_W.UnLoadGoods_Enable_B1=1 THEN
	Station_Status[3].UnLoadGoods_Enable:=TRUE;
ELSE
	Station_Status[3].UnLoadGoods_Enable:=FALSE;
END_IF;
IF Master_W.UnLoadGoods_Enable_B2=1 THEN
	Station_Status[4].UnLoadGoods_Enable:=TRUE;
ELSE
	Station_Status[4].UnLoadGoods_Enable:=FALSE;
END_IF;

(*Read*)
Master_R.Stacker_Status:=Auto_Data.Stacker_Status;
Master_R.Auto_Step:=Auto_Data.Auto_Step;
Master_R.Error_Code:=Auto_Data.Error_Code;
Master_R.Task_Status:=Auto_Data.Task_Status;
Master_R.Current_Task_ID:=Auto_Data.Current_Task_ID;
Master_R.Total_Number_Tasks:=Auto_Data.Total_Number_Tasks;
INT(1,Auto_Data.X_Current_Actual_Position ,Master_R.X_Current_Actual_Position  );
INT(1,Auto_Data.Y_Current_Actual_Position ,Master_R.Y_Current_Actual_Position  );
INT(1,Auto_Data.Z_Current_Actual_Position ,Master_R.Z_Current_Actual_Position  );
INT(1,Auto_Data.X_Current_Actual_Speed,Master_R.X_Current_Actual_Speed  );
INT(1,Auto_Data.Y_Current_Actual_Speed,Master_R.Y_Current_Actual_Speed  );
INT(1,Auto_Data.Z_Current_Actual_Speed,Master_R.Z_Current_Actual_Speed  );
Master_R.Current_Mode:=Mode;
Master_R.Heartbeat:=Master_W.Heartbeat;
Master_R.Step_Record:=Record.Auto_Step;
Master_R.X_Torque:=Axle_X_Sew_Read.Actual_Torque/10;
Master_R.Y_Torque:=Axle_Y_Sew_Read.Actual_Torque/10;
Master_R.Z_Torque:=Axle_Z_Sew_Read.Actual_Torque/10;
Master_R.X_Alarm_Code:=Axle_X_Alalm;
Master_R.Y_Alarm_Code:=Axle_Y_Alalm;
Master_R.Z_Alarm_Code:=Axle_Z_Alalm;
Master_R.Stacker_Current_Column:=Stacker_Current_Column;
Master_R.Stacker_Current_Layer:=Stacker_Current_Layer;
Master_R.Warning_Code:=Warning_Code;

(*堆垛机地面手动控制中*)
IF Stacker_W_Control_Bit.Apply_Manual_Control AND Manual_Mode THEN
	Stacker_R_Status_Bit.Stacker_A01ManualControl:=TRUE;
	
	Axle[0].Jog_Forward := Stacker_W_Control_Bit.X_Jog_Forward;
    Axle[0].Jog_Reverse :=Stacker_W_Control_Bit.X_Jog_Reverse;
    Axle[1].Jog_Forward  :=Stacker_W_Control_Bit.Y_Jog_Forward;
    Axle[1].Jog_Reverse  :=Stacker_W_Control_Bit.Y_Jog_Reverse;
    Axle[2].Jog_Forward  :=Stacker_W_Control_Bit.Z_Jog_Forward;
    Axle[2].Jog_Reverse  :=Stacker_W_Control_Bit.Z_Jog_Reverse;
    Manual_Y_Force_Enable:=Stacker_W_Control_Bit.Manual_Y_Force_Enable;
    Manual.Position_Coords_Switch:=Stacker_W_Control_Bit.Position_Coords_Switch;
    Manual.X_ManualStart_Position:=Stacker_W_Control_Bit.X_ManualStart_Position;
    Manual.Y_ManualStart_Position:=Stacker_W_Control_Bit.Y_ManualStart_Position;
    Manual.Z_ManualStart_Position:=Stacker_W_Control_Bit.Z_ManualStart_Position;
ELSE
	Stacker_R_Status_Bit.Stacker_A01ManualControl:=FALSE;
END_IF;

Stacker_R_Status_Bit.Fork_Zero:=Fork_Zero;
Stacker_R_Status_Bit.Advance_To_Position:=DInput.Walk_Forward_TO_Pos;
Stacker_R_Status_Bit.Retreat_To_Position:=DInput.Walk_Reverse_TO_Pos;
Stacker_R_Status_Bit.Ascend_To_Position:=DInput.Lift_Up_TO_Pos;
Stacker_R_Status_Bit.Descend_To_Position:=DInput.Lift_Down_TO_Pos;
Stacker_R_Status_Bit.Left_To_Position:=DInput.Fork_Left_To_Pos;
Stacker_R_Status_Bit.Right_To_Position:=DInput.Fork_Right_To_Pos;
END_PROGRAM

PROGRAM 02_IO
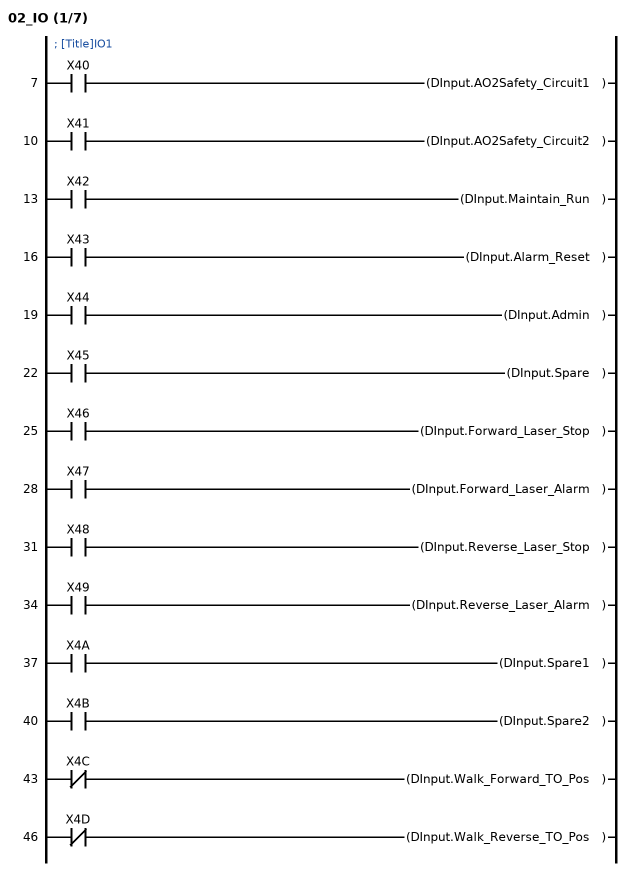
; [Title]IO1
7     LD      X40
      OUT     DInput.AO2Safety_Circuit1
10    LD      X41
      OUT     DInput.AO2Safety_Circuit2
13    LD      X42
      OUT     DInput.Maintain_Run
16    LD      X43
      OUT     DInput.Alarm_Reset
19    LD      X44
      OUT     DInput.Admin
22    LD      X45
      OUT     DInput.Spare
25    LD      X46
      OUT     DInput.Forward_Laser_Stop
28    LD      X47
      OUT     DInput.Forward_Laser_Alarm
31    LD      X48
      OUT     DInput.Reverse_Laser_Stop
34    LD      X49
      OUT     DInput.Reverse_Laser_Alarm
37    LD      X4A
      OUT     DInput.Spare1
40    LD      X4B
      OUT     DInput.Spare2
43    LDI     X4C
      OUT     DInput.Walk_Forward_TO_Pos
46    LDI     X4D
      OUT     DInput.Walk_Reverse_TO_Pos
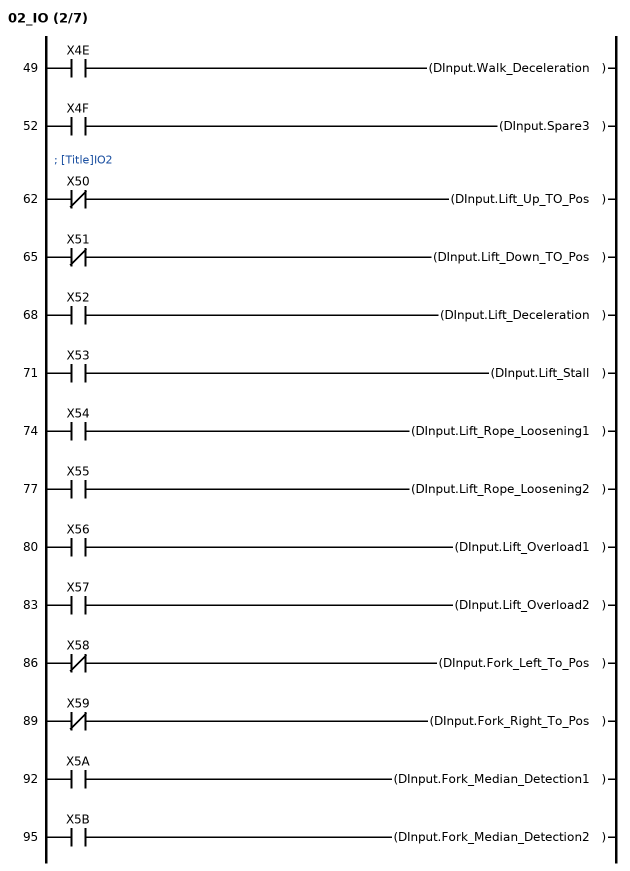
49    LD      X4E
      OUT     DInput.Walk_Deceleration
52    LD      X4F
      OUT     DInput.Spare3
; [Title]IO2
62    LDI     X50
      OUT     DInput.Lift_Up_TO_Pos
65    LDI     X51
      OUT     DInput.Lift_Down_TO_Pos
68    LD      X52
      OUT     DInput.Lift_Deceleration
71    LD      X53
      OUT     DInput.Lift_Stall
74    LD      X54
      OUT     DInput.Lift_Rope_Loosening1
77    LD      X55
      OUT     DInput.Lift_Rope_Loosening2
80    LD      X56
      OUT     DInput.Lift_Overload1
83    LD      X57
      OUT     DInput.Lift_Overload2
86    LDI     X58
      OUT     DInput.Fork_Left_To_Pos
89    LDI     X59
      OUT     DInput.Fork_Right_To_Pos
92    LD      X5A
      OUT     DInput.Fork_Median_Detection1
95    LD      X5B
      OUT     DInput.Fork_Median_Detection2
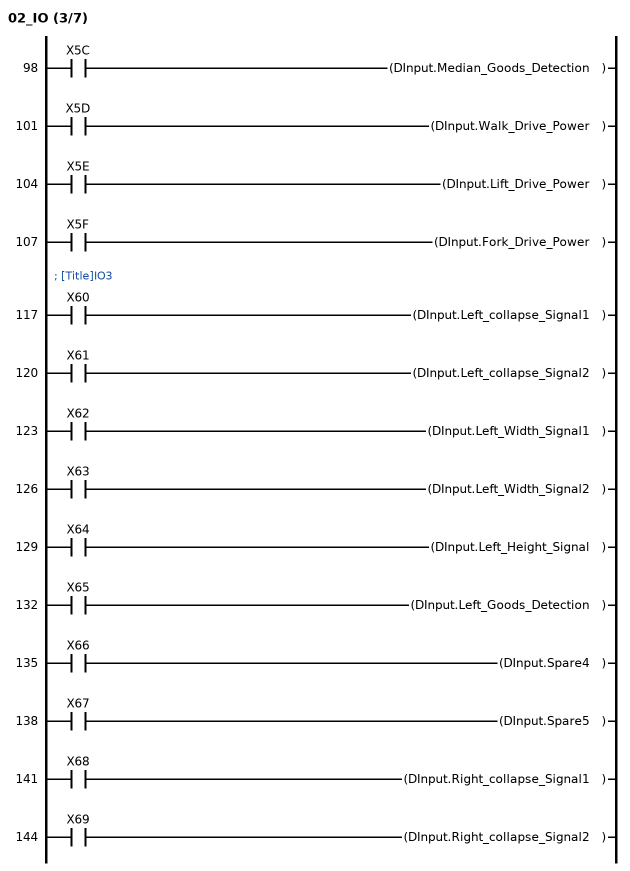
98    LD      X5C
      OUT     DInput.Median_Goods_Detection
101   LD      X5D
      OUT     DInput.Walk_Drive_Power
104   LD      X5E
      OUT     DInput.Lift_Drive_Power
107   LD      X5F
      OUT     DInput.Fork_Drive_Power
; [Title]IO3
117   LD      X60
      OUT     DInput.Left_collapse_Signal1
120   LD      X61
      OUT     DInput.Left_collapse_Signal2
123   LD      X62
      OUT     DInput.Left_Width_Signal1
126   LD      X63
      OUT     DInput.Left_Width_Signal2
129   LD      X64
      OUT     DInput.Left_Height_Signal
132   LD      X65
      OUT     DInput.Left_Goods_Detection
135   LD      X66
      OUT     DInput.Spare4
138   LD      X67
      OUT     DInput.Spare5
141   LD      X68
      OUT     DInput.Right_collapse_Signal1
144   LD      X69
      OUT     DInput.Right_collapse_Signal2
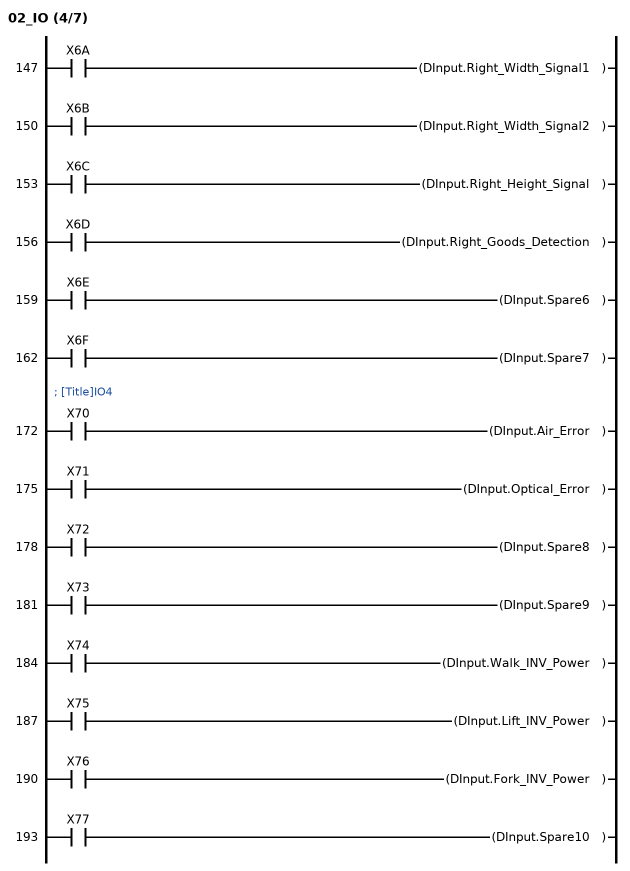
147   LD      X6A
      OUT     DInput.Right_Width_Signal1
150   LD      X6B
      OUT     DInput.Right_Width_Signal2
153   LD      X6C
      OUT     DInput.Right_Height_Signal
156   LD      X6D
      OUT     DInput.Right_Goods_Detection
159   LD      X6E
      OUT     DInput.Spare6
162   LD      X6F
      OUT     DInput.Spare7
; [Title]IO4
172   LD      X70
      OUT     DInput.Air_Error
175   LD      X71
      OUT     DInput.Optical_Error
178   LD      X72
      OUT     DInput.Spare8
181   LD      X73
      OUT     DInput.Spare9
184   LD      X74
      OUT     DInput.Walk_INV_Power
187   LD      X75
      OUT     DInput.Lift_INV_Power
190   LD      X76
      OUT     DInput.Fork_INV_Power
193   LD      X77
      OUT     DInput.Spare10
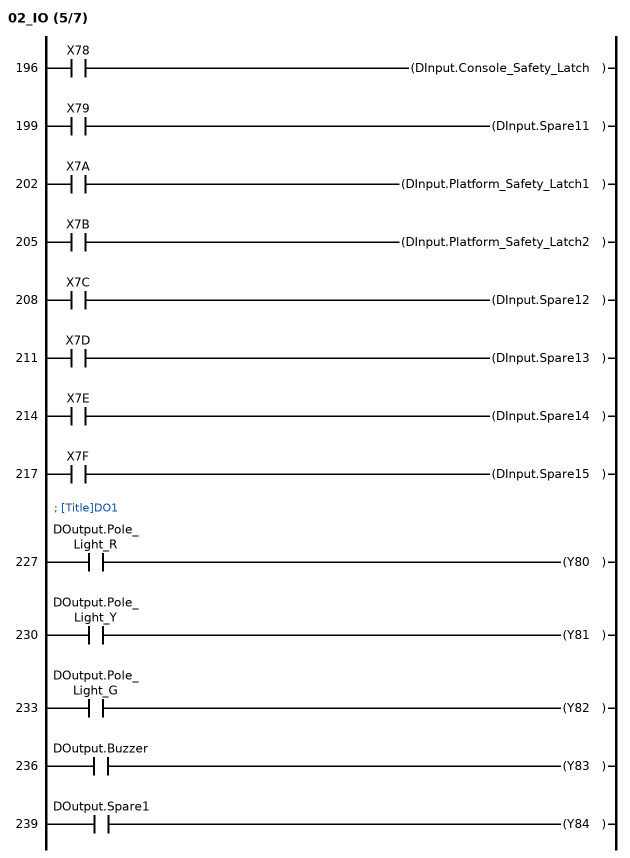
196   LD      X78
      OUT     DInput.Console_Safety_Latch
199   LD      X79
      OUT     DInput.Spare11
202   LD      X7A
      OUT     DInput.Platform_Safety_Latch1
205   LD      X7B
      OUT     DInput.Platform_Safety_Latch2
208   LD      X7C
      OUT     DInput.Spare12
211   LD      X7D
      OUT     DInput.Spare13
214   LD      X7E
      OUT     DInput.Spare14
217   LD      X7F
      OUT     DInput.Spare15
; [Title]DO1
227   LD      DOutput.Pole_Light_R
      OUT     Y80
230   LD      DOutput.Pole_Light_Y
      OUT     Y81
233   LD      DOutput.Pole_Light_G
      OUT     Y82
236   LD      DOutput.Buzzer
      OUT     Y83
239   LD      DOutput.Spare1
      OUT     Y84
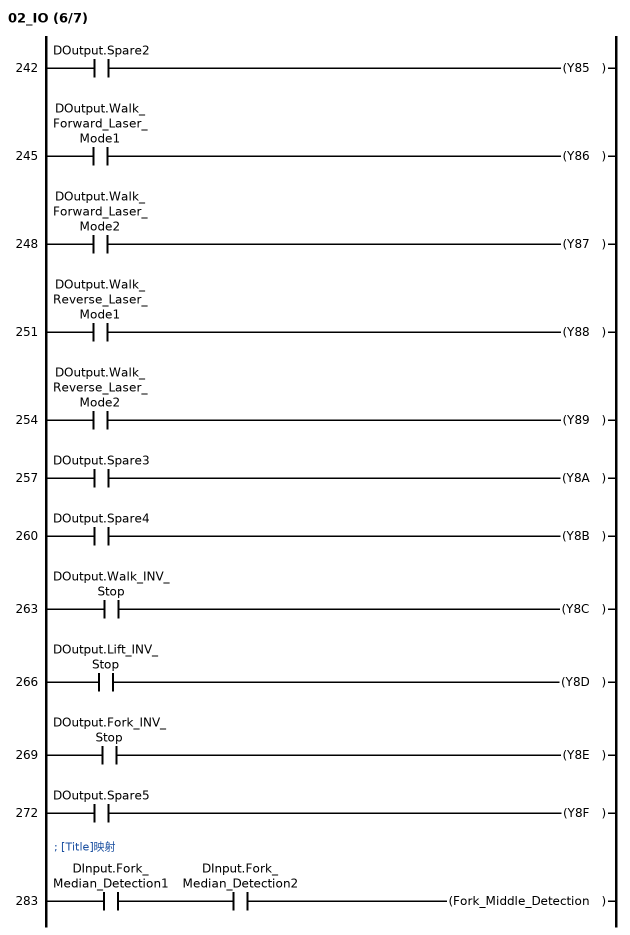
242   LD      DOutput.Spare2
      OUT     Y85
245   LD      DOutput.Walk_Forward_Laser_Mode1
      OUT     Y86
248   LD      DOutput.Walk_Forward_Laser_Mode2
      OUT     Y87
251   LD      DOutput.Walk_Reverse_Laser_Mode1
      OUT     Y88
254   LD      DOutput.Walk_Reverse_Laser_Mode2
      OUT     Y89
257   LD      DOutput.Spare3
      OUT     Y8A
260   LD      DOutput.Spare4
      OUT     Y8B
263   LD      DOutput.Walk_INV_Stop
      OUT     Y8C
266   LD      DOutput.Lift_INV_Stop
      OUT     Y8D
269   LD      DOutput.Fork_INV_Stop
      OUT     Y8E
272   LD      DOutput.Spare5
      OUT     Y8F
; [Title]映射
283   LD      DInput.Fork_Median_Detection1
      AND     DInput.Fork_Median_Detection2
      OUT     Fork_Middle_Detection
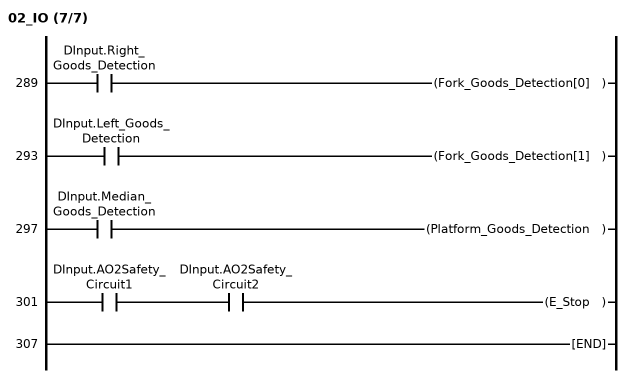
289   LD      DInput.Right_Goods_Detection
      OUT     Fork_Goods_Detection[0]
293   LD      DInput.Left_Goods_Detection
      OUT     Fork_Goods_Detection[1]
297   LD      DInput.Median_Goods_Detection
      OUT     Platform_Goods_Detection
301   LD      DInput.AO2Safety_Circuit1
      AND     DInput.AO2Safety_Circuit2
      OUT     E_Stop
307   END
END_PROGRAM
